C03632=1051.744,-43.846,429.339,170.450,30.999,155.847
C03633=1051.750,-43.595,429.326,170.452,31.001,155.847
C03634=1051.756,-43.346,429.313,170.454,31.002,155.847
C03635=1051.763,-43.096,429.301,170.456,31.005,155.847
C03636=1051.769,-42.847,429.288,170.458,31.006,155.848
C03637=1051.775,-42.597,429.275,170.460,31.008,155.848
C03638=1051.781,-42.347,429.262,170.461,31.009,155.848
C03639=1051.787,-42.098,429.249,170.463,31.011,155.848
C03640=1051.794,-41.848,429.237,170.465,31.012,155.848
C03641=1051.800,-41.599,429.224,170.467,31.014,155.848
C03642=1051.806,-41.349,429.211,170.469,31.015,155.849
C03643=1051.812,-41.100,429.198,170.471,31.017,155.849
C03644=1051.819,-40.849,429.185,170.473,31.018,155.849
C03645=1051.825,-40.600,429.172,170.475,31.020,155.849
C03646=1051.832,-40.351,429.160,170.476,31.021,155.849
C03647=1051.838,-40.101,429.147,170.478,31.023,155.849
C03648=1051.844,-39.852,429.133,170.480,31.024,155.850
C03649=1051.850,-39.602,429.121,170.482,31.026,155.850
C03650=1051.856,-39.353,429.108,170.484,31.028,155.850
C03651=1051.862,-39.103,429.095,170.486,31.030,155.850
C03652=1051.870,-38.853,429.082,170.488,31.031,155.850
C03653=1051.876,-38.604,429.069,170.490,31.033,155.850
C03654=1051.882,-38.354,429.056,170.491,31.034,155.851
C03655=1051.888,-38.105,429.043,170.493,31.036,155.851
C03656=1051.894,-37.855,429.030,170.495,31.037,155.851
C03657=1051.900,-37.606,429.017,170.497,31.039,155.851
C03658=1051.906,-37.357,429.004,170.499,31.041,155.851
C03659=1051.912,-37.107,428.991,170.501,31.042,155.852
C03660=1051.918,-36.856,428.977,170.503,31.044,155.852
C03661=1051.925,-36.607,428.964,170.504,31.046,155.852
C03662=1051.930,-36.357,428.951,170.506,31.048,155.852
C03663=1051.937,-36.108,428.938,170.508,31.049,155.852
C03664=1051.943,-35.859,428.925,170.509,31.051,155.853
C03665=1051.949,-35.609,428.912,170.511,31.053,155.853
C03666=1051.956,-35.359,428.899,170.513,31.054,155.853
C03667=1051.962,-35.080,428.884,170.516,31.056,155.853
C03668=1051.969,-34.799,428.869,170.518,31.058,155.853
C03669=1051.976,-34.519,428.855,170.519,31.060,155.854
C03670=1051.983,-34.239,428.840,170.521,31.062,155.854
C03671=1051.990,-33.989,428.826,170.523,31.063,155.854
C03672=1051.995,-33.739,428.813,170.525,31.065,155.854
C03673=1052.001,-33.490,428.800,170.527,31.067,155.854
C03674=1052.008,-33.241,428.786,170.529,31.068,155.855
C03675=1052.014,-32.991,428.773,170.531,31.070,155.855
C03676=1052.020,-32.741,428.760,170.533,31.072,155.855
C03677=1052.027,-32.492,428.747,170.534,31.074,155.855
C03678=1052.033,-32.242,428.734,170.536,31.075,155.855
C03679=1052.039,-31.993,428.720,170.538,31.077,155.856
C03680=1052.046,-31.743,428.707,170.540,31.079,155.856
C03681=1052.052,-31.494,428.694,170.542,31.080,155.856
C03682=1052.058,-31.244,428.681,170.544,31.082,155.856
C03683=1052.063,-30.994,428.667,170.546,31.084,155.856
C03684=1052.070,-30.744,428.653,170.547,31.085,155.857
C03685=1052.076,-30.495,428.640,170.548,31.087,155.857
C03686=1052.083,-30.246,428.627,170.550,31.088,155.857
C03687=1052.089,-29.997,428.614,170.552,31.091,155.857
C03688=1052.096,-29.747,428.600,170.554,31.092,155.857
C03689=1052.102,-29.497,428.587,170.556,31.094,155.858
C03690=1052.108,-29.247,428.574,170.558,31.096,155.858
C03691=1052.115,-28.997,428.561,170.560,31.097,155.858
C03692=1052.120,-28.748,428.547,170.561,31.099,155.858
C03693=1052.126,-28.499,428.533,170.563,31.101,155.858
C03694=1052.133,-28.249,428.520,170.565,31.102,155.859
C03695=1052.139,-27.999,428.507,170.567,31.104,155.859
C03696=1052.146,-27.750,428.493,170.569,31.106,155.859
C03697=1052.152,-27.501,428.480,170.571,31.108,155.859
C03698=1052.159,-27.251,428.466,170.573,31.109,155.859
C03699=1052.164,-27.001,428.453,170.575,31.111,155.860
C03700=1052.170,-26.752,428.439,170.575,31.113,155.860
C03701=1052.177,-26.502,428.426,170.577,31.114,155.860
C03702=1052.183,-26.253,428.412,170.579,31.116,155.860
C03703=1052.189,-26.003,428.398,170.581,31.118,155.861
C03704=1052.196,-25.753,428.385,170.583,31.120,155.861
C03705=1052.201,-25.504,428.371,170.585,31.121,155.861
C03706=1052.207,-25.254,428.358,170.587,31.124,155.861
C03707=1052.214,-25.004,428.344,170.589,31.125,155.861
C03708=1052.220,-24.755,428.330,170.590,31.127,155.862
C03709=1052.226,-24.506,428.317,170.592,31.129,155.862
C03710=1052.232,-24.256,428.304,170.594,31.130,155.862
C03711=1052.238,-24.006,428.289,170.595,31.132,155.862
C03712=1052.245,-23.757,428.275,170.597,31.134,155.863
C03713=1052.250,-23.508,428.262,170.599,31.136,155.863
C03714=1052.257,-23.258,428.248,170.601,31.137,155.863
C03715=1052.263,-23.009,428.235,170.603,31.140,155.863
C03716=1052.269,-22.758,428.220,170.604,31.141,155.863
C03717=1052.275,-22.509,428.207,170.606,31.143,155.864
C03718=1052.282,-22.260,428.194,170.608,31.145,155.864
C03719=1052.288,-22.010,428.179,170.610,31.147,155.864
C03720=1052.294,-21.761,428.166,170.612,31.148,155.864
C03721=1052.300,-21.511,428.152,170.613,31.150,155.865
C03722=1052.307,-21.261,428.138,170.615,31.152,155.865
C03723=1052.313,-21.012,428.125,170.616,31.154,155.865
C03724=1052.319,-20.762,428.111,170.618,31.155,155.865
C03725=1052.325,-20.513,428.097,170.620,31.158,155.866
C03726=1052.331,-20.264,428.083,170.622,31.159,155.866
C03727=1052.338,-20.014,428.069,170.624,31.161,155.866
C03728=1052.344,-19.764,428.056,170.626,31.163,155.866
C03729=1052.350,-19.515,428.041,170.628,31.165,155.866
C03730=1052.356,-19.265,428.028,170.630,31.166,155.867
C03731=1052.363,-18.984,428.012,170.631,31.169,155.867
C03732=1052.370,-18.703,427.996,170.633,31.171,155.867
C03733=1052.377,-18.422,427.981,170.635,31.173,155.867
C03734=1052.385,-18.141,427.965,170.637,31.175,155.868
C03735=1052.390,-17.892,427.951,170.639,31.176,155.868
C03736=1052.397,-17.643,427.938,170.641,31.179,155.868
C03737=1052.403,-17.393,427.923,170.643,31.180,155.868
C03738=1052.409,-17.144,427.910,170.644,31.182,155.869
C03739=1052.416,-16.894,427.895,170.645,31.184,155.869
C03740=1052.422,-16.645,427.882,170.647,31.186,155.869
C03741=1052.429,-16.395,427.868,170.649,31.187,155.869
C03742=1052.434,-16.146,427.854,170.651,31.189,155.870
C03743=1052.441,-15.896,427.840,170.653,31.191,155.870
C03744=1052.447,-15.646,427.826,170.655,31.193,155.870
C03745=1052.454,-15.397,427.812,170.657,31.195,155.870
C03746=1052.459,-15.147,427.798,170.658,31.197,155.870
C03747=1052.466,-14.897,427.784,170.660,31.198,155.871
C03748=1052.472,-14.648,427.770,170.661,31.200,155.871
C03749=1052.478,-14.398,427.755,170.663,31.202,155.871
C03750=1052.484,-14.149,427.741,170.665,31.204,155.871
C03751=1052.491,-13.899,427.727,170.667,31.206,155.872
C03752=1052.496,-13.650,427.713,170.669,31.208,155.872
C03753=1052.503,-13.400,427.699,170.671,31.210,155.872
C03754=1052.509,-13.151,427.685,170.672,31.212,155.872
C03755=1052.515,-12.901,427.670,170.673,31.214,155.873
C03756=1052.521,-12.652,427.657,170.675,31.215,155.873
C03757=1052.528,-12.402,427.642,170.677,31.217,155.873
C03758=1052.533,-12.153,427.628,170.679,31.219,155.873
C03759=1052.540,-11.903,427.614,170.681,31.221,155.874
C03760=1052.546,-11.654,427.600,170.683,31.223,155.874
C03761=1052.552,-11.404,427.585,170.685,31.225,155.874
C03762=1052.558,-11.155,427.572,170.685,31.227,155.874
C03763=1052.565,-10.905,427.557,170.687,31.229,155.875
C03764=1052.570,-10.655,427.543,170.689,31.231,155.875
C03765=1052.577,-10.406,427.529,170.691,31.232,155.875
C03766=1052.583,-10.157,427.514,170.693,31.234,155.875
C03767=1052.589,-9.907,427.500,170.695,31.237,155.876
C03768=1052.596,-9.658,427.486,170.697,31.238,155.876
C03769=1052.602,-9.408,427.471,170.698,31.240,155.876
C03770=1052.608,-9.158,427.457,170.699,31.242,155.876
C03771=1052.614,-8.909,427.443,170.701,31.244,155.877
C03772=1052.621,-8.659,427.428,170.703,31.246,155.877
C03773=1052.626,-8.410,427.414,170.705,31.248,155.877
C03774=1052.633,-8.160,427.400,170.707,31.250,155.877
C03775=1052.639,-7.912,427.386,170.708,31.251,155.878
C03776=1052.645,-7.662,427.371,170.710,31.253,155.878
C03777=1052.652,-7.412,427.356,170.712,31.256,155.878
C03778=1052.658,-7.163,427.342,170.713,31.257,155.878
C03779=1052.664,-6.913,427.328,170.715,31.259,155.879
C03780=1052.670,-6.663,427.313,170.717,31.261,155.879
C03781=1052.676,-6.414,427.299,170.718,31.263,155.879
C03782=1052.683,-6.164,427.285,170.720,31.265,155.879
C03783=1052.689,-5.915,427.270,170.722,31.267,155.880
C03784=1052.695,-5.665,427.255,170.724,31.268,155.880
C03785=1052.702,-5.416,427.240,170.726,31.271,155.880
C03786=1052.708,-5.167,427.227,170.727,31.273,155.880
C03787=1052.714,-4.917,427.212,170.729,31.275,155.881
C03788=1052.721,-4.667,427.197,170.730,31.276,155.881
C03789=1052.727,-4.418,427.184,170.732,31.278,155.881
C03790=1052.733,-4.168,427.169,170.734,31.280,155.881
C03791=1052.740,-3.919,427.154,170.736,31.282,155.882
C03792=1052.745,-3.670,427.140,170.738,31.284,155.882
C03793=1052.752,-3.420,427.126,170.739,31.286,155.882
C03794=1052.759,-3.170,427.111,170.740,31.288,155.883
C03795=1052.765,-2.888,427.094,170.742,31.290,155.883
C03796=1052.772,-2.606,427.078,170.744,31.292,155.883
C03797=1052.779,-2.323,427.062,170.746,31.294,155.883
C03798=1052.786,-2.040,427.045,170.749,31.297,155.884
C03799=1052.792,-1.791,427.030,170.750,31.299,155.884
C03800=1052.797,-1.541,427.014,170.752,31.301,155.884
C03801=1052.804,-1.292,426.999,170.753,31.303,155.885
C03802=1052.810,-1.043,426.985,170.755,31.305,155.885
C03803=1052.816,-0.793,426.970,170.757,31.307,155.885
C03804=1052.822,-0.543,426.956,170.758,31.309,155.885
C03805=1052.828,-0.294,426.941,170.760,31.311,155.886
C03806=1052.834,-0.044,426.926,170.762,31.313,155.886
C03807=1052.841,0.206,426.911,170.764,31.315,155.886
C03808=1052.846,0.455,426.897,170.765,31.318,155.887
C03809=1052.853,0.704,426.882,170.766,31.319,155.887
C03810=1052.859,0.954,426.867,170.768,31.321,155.887
C03811=1052.865,1.203,426.852,170.770,31.323,155.887
C03812=1052.871,1.452,426.837,170.772,31.325,155.888
C03813=1052.878,1.702,426.822,170.774,31.327,155.888
C03814=1052.883,1.951,426.808,170.775,31.329,155.888
C03815=1052.890,2.201,426.793,170.777,31.331,155.888
C03816=1052.896,2.450,426.778,170.778,31.334,155.889
C03817=1052.902,2.699,426.763,170.780,31.336,155.889
C03818=1052.908,2.949,426.748,170.782,31.337,155.889
C03819=1052.915,3.199,426.733,170.783,31.339,155.890
C03820=1052.920,3.449,426.718,170.785,31.341,155.890
C03821=1052.926,3.698,426.703,170.787,31.343,155.890
C03822=1052.933,3.947,426.688,170.789,31.345,155.890
C03823=1052.939,4.197,426.673,170.790,31.347,155.891
C03824=1052.945,4.447,426.658,170.792,31.350,155.891
C03825=1052.951,4.695,426.644,170.793,31.352,155.891
C03826=1052.958,4.945,426.629,170.795,31.354,155.892
C03827=1052.964,5.195,426.614,170.797,31.355,155.892
C03828=1052.970,5.444,426.599,170.798,31.357,155.892
C03829=1052.976,5.693,426.584,170.800,31.359,155.892
C03830=1052.982,5.943,426.569,170.802,31.361,155.893
C03831=1052.989,6.193,426.555,170.804,31.364,155.893
C03832=1052.995,6.443,426.539,170.805,31.366,155.893
C03833=1053.001,6.691,426.524,170.806,31.368,155.893
C03834=1053.007,6.941,426.509,170.808,31.370,155.894
C03835=1053.013,7.190,426.494,170.810,31.372,155.894
C03836=1053.020,7.440,426.479,170.812,31.374,155.894
C03837=1053.026,7.690,426.464,170.813,31.375,155.895
C03838=1053.033,7.939,426.449,170.815,31.377,155.895
C03839=1053.038,8.188,426.434,170.817,31.380,155.895
C03840=1053.045,8.437,426.419,170.819,31.382,155.895
C03841=1053.051,8.687,426.403,170.820,31.384,155.896
C03842=1053.057,8.937,426.388,170.821,31.386,155.896
C03843=1053.063,9.187,426.373,170.823,31.388,155.896
C03844=1053.070,9.436,426.358,170.825,31.390,155.897
C03845=1053.076,9.685,426.344,170.827,31.392,155.897
C03846=1053.082,9.934,426.328,170.829,31.394,155.897
C03847=1053.089,10.184,426.313,170.830,31.396,155.897
C03848=1053.095,10.434,426.298,170.832,31.398,155.898
C03849=1053.101,10.684,426.283,170.833,31.400,155.898
C03850=1053.107,10.933,426.267,170.835,31.402,155.898
C03851=1053.114,11.182,426.252,170.836,31.404,155.899
C03852=1053.120,11.431,426.237,170.838,31.406,155.899
C03853=1053.126,11.681,426.223,170.840,31.408,155.899
C03854=1053.133,11.930,426.207,170.842,31.410,155.899
C03855=1053.139,12.180,426.192,170.844,31.412,155.900
C03856=1053.145,12.429,426.176,170.845,31.414,155.900
C03857=1053.151,12.679,426.161,170.846,31.416,155.900
C03858=1053.158,12.928,426.146,170.848,31.418,155.900
C03859=1053.165,13.213,426.128,170.850,31.421,155.901
C03860=1053.172,13.497,426.111,170.852,31.423,155.901
C03861=1053.179,13.781,426.094,170.854,31.425,155.901
C03862=1053.186,14.066,426.077,170.856,31.427,155.902
C03863=1053.193,14.315,426.061,170.858,31.429,155.902
C03864=1053.199,14.565,426.046,170.859,31.431,155.902
C03865=1053.205,14.814,426.030,170.860,31.434,155.903
C03866=1053.211,15.064,426.015,170.862,31.436,155.903
C03867=1053.217,15.314,426.000,170.864,31.438,155.903
C03868=1053.224,15.563,425.984,170.865,31.440,155.904
C03869=1053.230,15.813,425.969,170.867,31.442,155.904
C03870=1053.236,16.062,425.953,170.869,31.444,155.904
C03871=1053.243,16.311,425.938,170.871,31.446,155.904
C03872=1053.248,16.561,425.923,170.872,31.448,155.905
C03873=1053.254,16.810,425.907,170.873,31.450,155.905
C03874=1053.260,17.060,425.892,170.875,31.452,155.905
C03875=1053.267,17.309,425.876,170.877,31.454,155.906
C03876=1053.273,17.558,425.861,170.878,31.456,155.906
C03877=1053.279,17.808,425.845,170.880,31.458,155.906
C03878=1053.285,18.057,425.830,170.882,31.461,155.906
C03879=1053.291,18.307,425.814,170.884,31.463,155.907
C03880=1053.298,18.556,425.799,170.885,31.465,155.907
C03881=1053.304,18.805,425.783,170.887,31.467,155.907
C03882=1053.310,19.055,425.767,170.888,31.469,155.908
C03883=1053.317,19.304,425.752,170.890,31.471,155.908
C03884=1053.322,19.554,425.736,170.891,31.473,155.908
C03885=1053.329,19.803,425.720,170.893,31.475,155.909
C03886=1053.335,20.053,425.706,170.895,31.477,155.909
C03887=1053.341,20.302,425.689,170.897,31.479,155.909
C03888=1053.347,20.552,425.673,170.898,31.481,155.909
C03889=1053.354,20.801,425.658,170.900,31.484,155.910
C03890=1053.360,21.051,425.642,170.901,31.486,155.910
C03891=1053.366,21.300,425.627,170.903,31.488,155.910
C03892=1053.372,21.550,425.611,170.904,31.490,155.911
C03893=1053.379,21.799,425.595,170.906,31.492,155.911
C03894=1053.384,22.049,425.579,170.908,31.494,155.911
C03895=1053.391,22.298,425.564,170.909,31.496,155.912
C03896=1053.397,22.548,425.548,170.911,31.498,155.912
C03897=1053.403,22.797,425.533,170.913,31.500,155.912
C03898=1053.409,23.046,425.516,170.914,31.502,155.913
C03899=1053.416,23.296,425.501,170.915,31.505,155.913
C03900=1053.422,23.545,425.485,170.917,31.507,155.913
C03901=1053.428,23.794,425.469,170.919,31.509,155.914
C03902=1053.434,24.044,425.454,170.921,31.511,155.914
C03903=1053.440,24.293,425.438,170.922,31.513,155.914
C03904=1053.447,24.542,425.422,170.924,31.515,155.914
C03905=1053.452,24.792,425.406,170.926,31.517,155.915
C03906=1053.459,25.041,425.391,170.928,31.519,155.915
C03907=1053.465,25.291,425.375,170.928,31.521,155.915
C03908=1053.471,25.540,425.358,170.930,31.524,155.916
C03909=1053.477,25.790,425.343,170.932,31.526,155.916
C03910=1053.483,26.039,425.327,170.933,31.528,155.916
C03911=1053.490,26.288,425.311,170.935,31.530,155.917
C03912=1053.496,26.538,425.295,170.937,31.532,155.917
C03913=1053.502,26.787,425.280,170.939,31.534,155.917
C03914=1053.508,27.037,425.264,170.940,31.536,155.917
C03915=1053.514,27.286,425.248,170.942,31.539,155.918
C03916=1053.521,27.535,425.232,170.943,31.541,155.918
C03917=1053.527,27.785,425.215,170.944,31.543,155.918
C03918=1053.533,28.035,425.200,170.946,31.545,155.919
C03919=1053.540,28.284,425.184,170.948,31.547,155.919
C03920=1053.546,28.533,425.168,170.950,31.549,155.919
C03921=1053.552,28.783,425.152,170.951,31.551,155.920
C03922=1053.558,29.032,425.136,170.953,31.554,155.920
C03923=1053.565,29.317,425.118,170.955,31.556,155.920
C03924=1053.573,29.603,425.099,170.956,31.558,155.921
C03925=1053.579,29.889,425.081,170.958,31.561,155.921
C03926=1053.586,30.175,425.063,170.960,31.564,155.921
C03927=1053.592,30.424,425.046,170.962,31.566,155.922
C03928=1053.598,30.673,425.030,170.963,31.568,155.922
C03929=1053.604,30.923,425.014,170.965,31.570,155.922
C03930=1053.611,31.172,424.998,170.967,31.573,155.923
C03931=1053.617,31.422,424.982,170.968,31.574,155.923
C03932=1053.623,31.672,424.966,170.969,31.577,155.923
C03933=1053.629,31.921,424.950,170.971,31.579,155.924
C03934=1053.635,32.170,424.933,170.973,31.581,155.924
C03935=1053.641,32.419,424.918,170.974,31.583,155.924
C03936=1053.647,32.669,424.902,170.976,31.585,155.925
C03937=1053.653,32.918,424.885,170.978,31.588,155.925
C03938=1053.660,33.168,424.869,170.979,31.589,155.925
C03939=1053.665,33.417,424.853,170.981,31.592,155.926
C03940=1053.672,33.665,424.836,170.983,31.594,155.926
C03941=1053.678,33.915,424.820,170.984,31.596,155.926
C03942=1053.684,34.164,424.804,170.985,31.598,155.927
C03943=1053.691,34.412,424.787,170.987,31.600,155.927
C03944=1053.697,34.662,424.771,170.989,31.602,155.927
C03945=1053.702,34.910,424.755,170.990,31.604,155.927
C03946=1053.709,35.159,424.740,170.992,31.607,155.928
C03947=1053.715,35.408,424.723,170.994,31.609,155.928
C03948=1053.722,35.658,424.706,170.995,31.611,155.928
C03949=1053.728,35.907,424.690,170.997,31.613,155.929
C03950=1053.734,36.157,424.674,170.998,31.615,155.929
C03951=1053.741,36.406,424.658,171.000,31.617,155.929
C03952=1053.747,36.655,424.642,171.001,31.620,155.930
C03953=1053.753,36.905,424.625,171.003,31.622,155.930
C03954=1053.759,37.155,424.609,171.005,31.624,155.930
C03955=1053.765,37.404,424.593,171.006,31.626,155.931
C03956=1053.771,37.653,424.576,171.008,31.628,155.931
C03957=1053.777,37.903,424.560,171.010,31.631,155.931
C03958=1053.784,38.152,424.543,171.011,31.633,155.932
C03959=1053.790,38.401,424.526,171.012,31.635,155.932
C03960=1053.796,38.651,424.510,171.014,31.637,155.932
C03961=1053.802,38.900,424.494,171.016,31.640,155.933
C03962=1053.808,39.149,424.478,171.017,31.642,155.933
C03963=1053.814,39.399,424.460,171.019,31.644,155.933
C03964=1053.820,39.648,424.444,171.021,31.646,155.934
C03965=1053.826,39.898,424.428,171.022,31.648,155.934
C03966=1053.832,40.147,424.412,171.024,31.650,155.934
C03967=1053.838,40.396,424.395,171.026,31.653,155.935
C03968=1053.845,40.646,424.378,171.026,31.655,155.935
C03969=1053.851,40.895,424.362,171.028,31.657,155.935
C03970=1053.857,41.144,424.345,171.030,31.659,155.936
C03971=1053.863,41.394,424.329,171.031,31.662,155.936
C03972=1053.870,41.643,424.312,171.033,31.664,155.936
C03973=1053.876,41.892,424.296,171.035,31.666,155.937
C03974=1053.882,42.142,424.279,171.036,31.668,155.937
C03975=1053.888,42.391,424.262,171.038,31.671,155.937
C03976=1053.894,42.641,424.246,171.040,31.673,155.938
C03977=1053.900,42.890,424.229,171.041,31.675,155.938
C03978=1053.906,43.140,424.213,171.042,31.677,155.938
C03979=1053.912,43.389,424.195,171.044,31.679,155.939
C03980=1053.918,43.638,424.179,171.046,31.681,155.939
C03981=1053.924,43.888,424.163,171.047,31.683,155.939
C03982=1053.931,44.136,424.146,171.049,31.686,155.940
C03983=1053.936,44.387,424.129,171.051,31.688,155.940
C03984=1053.943,44.636,424.112,171.052,31.691,155.940
C03985=1053.949,44.885,424.095,171.054,31.693,155.941
C03986=1053.955,45.134,424.079,171.056,31.695,155.941
C03987=1053.961,45.421,424.060,171.057,31.698,155.941
C03988=1053.969,45.707,424.040,171.058,31.700,155.942
C03989=1053.975,45.994,424.020,171.060,31.703,155.942
C03990=1053.982,46.281,424.001,171.062,31.705,155.943
C03991=1053.988,46.530,423.985,171.064,31.708,155.943
C03992=1053.994,46.780,423.967,171.066,31.710,155.943
C03993=1054.000,47.029,423.951,171.067,31.712,155.944
C03994=1054.006,47.278,423.934,171.069,31.715,155.944
C03995=1054.012,47.528,423.916,171.070,31.717,155.944
C03996=1054.019,47.777,423.899,171.071,31.719,155.945
C03997=1054.024,48.026,423.883,171.073,31.722,155.945
C03998=1054.031,48.275,423.866,171.075,31.724,155.945
C03999=1054.037,48.525,423.849,171.076,31.726,155.946
C04000=1054.043,48.774,423.832,171.078,31.728,155.946
C04001=1054.049,49.023,423.816,171.080,31.730,155.946
C04002=1054.055,49.273,423.798,171.081,31.733,155.947
C04003=1054.061,49.522,423.782,171.083,31.735,155.947
C04004=1054.067,49.771,423.765,171.085,31.737,155.947
C04005=1054.073,50.022,423.747,171.085,31.740,155.948
C04006=1054.079,50.270,423.730,171.087,31.742,155.948
C04007=1054.085,50.520,423.714,171.089,31.744,155.948
C04008=1054.091,50.769,423.696,171.090,31.746,155.949
C04009=1054.097,51.018,423.679,171.092,31.748,155.949
C04010=1054.104,51.268,423.663,171.094,31.751,155.950
C04011=1054.110,51.517,423.645,171.095,31.753,155.950
C04012=1054.115,51.767,423.629,171.097,31.755,155.950
C04013=1054.122,52.016,423.611,171.099,31.758,155.951
C04014=1054.128,52.265,423.594,171.099,31.760,155.951
C04015=1054.134,52.514,423.578,171.101,31.762,155.951
C04016=1054.141,52.764,423.560,171.103,31.764,155.952
C04017=1054.146,53.013,423.543,171.104,31.766,155.952
C04018=1054.153,53.263,423.526,171.106,31.768,155.952
C04019=1054.158,53.512,423.509,171.108,31.771,155.953
C04020=1054.165,53.761,423.492,171.109,31.773,155.953
C04021=1054.171,54.011,423.475,171.111,31.775,155.953
C04022=1054.177,54.260,423.457,171.113,31.778,155.954
C04023=1054.183,54.509,423.440,171.115,31.780,155.954
C04024=1054.189,54.759,423.424,171.115,31.782,155.954
C04025=1054.196,55.008,423.406,171.117,31.785,155.955
C04026=1054.202,55.257,423.389,171.119,31.787,155.955
C04027=1054.207,55.507,423.372,171.120,31.789,155.955
C04028=1054.214,55.756,423.355,171.122,31.791,155.956
C04029=1054.220,56.005,423.338,171.124,31.793,155.956
C04030=1054.226,56.255,423.320,171.125,31.796,155.956
C04031=1054.232,56.504,423.304,171.127,31.798,155.957
C04032=1054.239,56.753,423.286,171.129,31.800,155.957
C04033=1054.245,57.002,423.269,171.130,31.803,155.957
C04034=1054.251,57.252,423.251,171.131,31.805,155.958
C04035=1054.257,57.501,423.234,171.133,31.807,155.958
C04036=1054.263,57.751,423.217,171.134,31.809,155.958
C04037=1054.270,58.000,423.200,171.136,31.811,155.959
C04038=1054.276,58.249,423.182,171.138,31.813,155.959
C04039=1054.282,58.498,423.165,171.139,31.816,155.959
C04040=1054.288,58.748,423.148,171.141,31.818,155.960
C04041=1054.294,58.997,423.131,171.143,31.820,155.960
C04042=1054.301,59.247,423.114,171.144,31.822,155.960
C04043=1054.307,59.496,423.096,171.146,31.825,155.961
C04044=1054.313,59.745,423.079,171.147,31.827,155.961
C04045=1054.319,59.994,423.061,171.148,31.829,155.961
C04046=1054.325,60.244,423.045,171.150,31.831,155.962
C04047=1054.331,60.493,423.027,171.152,31.833,155.962
C04048=1054.338,60.743,423.010,171.153,31.835,155.962
C04049=1054.344,60.991,422.993,171.155,31.838,155.963
C04050=1054.350,61.241,422.975,171.157,31.840,155.963
C04051=1054.358,61.527,422.955,171.159,31.843,155.964
C04052=1054.365,61.811,422.935,171.161,31.845,155.964
C04053=1054.372,62.097,422.915,171.163,31.848,155.964
C04054=1054.379,62.383,422.896,171.163,31.850,155.965
C04055=1054.385,62.632,422.878,171.165,31.852,155.965
C04056=1054.392,62.881,422.861,171.167,31.855,155.965
C04057=1054.398,63.131,422.843,171.169,31.857,155.966
C04058=1054.404,63.380,422.826,171.170,31.859,155.966
C04059=1054.410,63.630,422.808,171.172,31.861,155.966
C04060=1054.416,63.878,422.791,171.174,31.864,155.967
C04061=1054.423,64.128,422.774,171.175,31.865,155.967
C04062=1054.429,64.377,422.756,171.177,31.868,155.967
C04063=1054.435,64.626,422.738,171.179,31.870,155.968
C04064=1054.442,64.876,422.721,171.180,31.872,155.968
C04065=1054.447,65.125,422.703,171.181,31.875,155.968
C04066=1054.453,65.375,422.685,171.183,31.877,155.969
C04067=1054.459,65.624,422.668,171.184,31.879,155.969
C04068=1054.466,65.873,422.651,171.186,31.881,155.970
C04069=1054.471,66.122,422.633,171.188,31.884,155.970
C04070=1054.478,66.371,422.614,171.189,31.886,155.970
C04071=1054.485,66.621,422.597,171.191,31.888,155.971
C04072=1054.490,66.870,422.579,171.193,31.891,155.971
C04073=1054.496,67.120,422.562,171.194,31.893,155.971
C04074=1054.502,67.368,422.545,171.196,31.895,155.972
C04075=1054.509,67.618,422.527,171.197,31.897,155.972
C04076=1054.515,67.868,422.509,171.198,31.899,155.972
C04077=1054.520,68.117,422.491,171.200,31.902,155.973
C04078=1054.527,68.366,422.474,171.202,31.904,155.973
C04079=1054.533,68.615,422.455,171.203,31.907,155.973
C04080=1054.539,68.864,422.438,171.205,31.909,155.974
C04081=1054.545,69.114,422.420,171.207,31.911,155.974
C04082=1054.551,69.363,422.403,171.208,31.913,155.974
C04083=1054.558,69.613,422.385,171.210,31.915,155.975
C04084=1054.564,69.862,422.367,171.212,31.918,155.975
C04085=1054.569,70.111,422.348,171.213,31.920,155.976
C04086=1054.576,70.360,422.331,171.214,31.923,155.976
C04087=1054.582,70.609,422.314,171.216,31.925,155.976
C04088=1054.588,70.859,422.296,171.217,31.927,155.977
C04089=1054.594,71.108,422.277,171.219,31.929,155.977
C04090=1054.600,71.357,422.259,171.221,31.932,155.977
C04091=1054.606,71.607,422.242,171.222,31.934,155.978
C04092=1054.612,71.857,422.224,171.224,31.937,155.978
C04093=1054.618,72.105,422.205,171.226,31.939,155.978
C04094=1054.624,72.355,422.187,171.227,31.941,155.979
C04095=1054.630,72.603,422.170,171.229,31.943,155.979
C04096=1054.637,72.853,422.152,171.231,31.946,155.980
C04097=1054.643,73.102,422.134,171.231,31.948,155.980
C04098=1054.648,73.351,422.116,171.233,31.950,155.980
C04099=1054.655,73.601,422.098,171.235,31.953,155.981
C04100=1054.661,73.850,422.080,171.236,31.955,155.981
C04101=1054.667,74.099,422.062,171.238,31.957,155.981
C04102=1054.673,74.348,422.043,171.240,31.959,155.982
C04103=1054.679,74.598,422.026,171.241,31.962,155.982
C04104=1054.685,74.848,422.008,171.243,31.964,155.982
C04105=1054.691,75.096,421.989,171.245,31.966,155.983
C04106=1054.697,75.346,421.971,171.246,31.968,155.983
C04107=1054.704,75.595,421.954,171.248,31.971,155.983
C04108=1054.710,75.844,421.936,171.249,31.973,155.984
C04109=1054.716,76.094,421.918,171.250,31.976,155.984
C04110=1054.722,76.343,421.899,171.252,31.978,155.985
C04111=1054.728,76.592,421.882,171.254,31.980,155.985
C04112=1054.734,76.842,421.864,171.255,31.982,155.985
C04113=1054.740,77.091,421.845,171.257,31.985,155.986
C04114=1054.747,77.340,421.827,171.259,31.987,155.986
C04115=1054.753,77.625,421.807,171.261,31.990,155.986
C04116=1054.760,77.911,421.786,171.262,31.992,155.987
C04117=1054.767,78.196,421.765,171.264,31.995,155.987
C04118=1054.774,78.481,421.744,171.266,31.997,155.988
C04119=1054.781,78.730,421.726,171.267,32.000,155.988
C04120=1054.786,78.979,421.708,171.269,32.002,155.988
C04121=1054.792,79.229,421.689,171.270,32.005,155.989
C04122=1054.798,79.478,421.670,171.272,32.007,155.989
C04123=1054.804,79.728,421.652,171.274,32.009,155.990
C04124=1054.810,79.976,421.634,171.275,32.011,155.990
C04125=1054.816,80.226,421.616,171.277,32.014,155.990
C04126=1054.823,80.475,421.597,171.279,32.016,155.991
C04127=1054.828,80.724,421.579,171.280,32.019,155.991
C04128=1054.834,80.973,421.560,171.282,32.021,155.991
C04129=1054.840,81.223,421.543,171.284,32.023,155.992
C04130=1054.847,81.472,421.524,171.284,32.026,155.992
C04131=1054.852,81.721,421.506,171.286,32.028,155.992
C04132=1054.859,81.970,421.488,171.288,32.031,155.993
C04133=1054.864,82.220,421.468,171.289,32.032,155.993
C04134=1054.871,82.469,421.450,171.291,32.035,155.994
C04135=1054.877,82.719,421.432,171.293,32.037,155.994
C04136=1054.883,82.967,421.414,171.294,32.040,155.994
C04137=1054.889,83.217,421.396,171.296,32.042,155.995
C04138=1054.894,83.466,421.376,171.298,32.044,155.995
C04139=1054.901,83.715,421.358,171.299,32.046,155.995
C04140=1054.906,83.965,421.340,171.301,32.049,155.996
C04141=1054.913,84.214,421.322,171.303,32.051,155.996
C04142=1054.919,84.463,421.303,171.303,32.054,155.997
C04143=1054.925,84.712,421.284,171.305,32.056,155.997
C04144=1054.931,84.962,421.266,171.307,32.058,155.997
C04145=1054.937,85.211,421.247,171.308,32.061,155.998
C04146=1054.943,85.459,421.229,171.310,32.063,155.998
C04147=1054.949,85.709,421.211,171.312,32.065,155.998
C04148=1054.955,85.959,421.192,171.313,32.067,155.999
C04149=1054.961,86.208,421.173,171.315,32.070,155.999
C04150=1054.968,86.457,421.154,171.317,32.072,155.999
C04151=1054.974,86.707,421.136,171.318,32.075,156.000
C04152=1054.979,86.955,421.117,171.320,32.077,156.000
C04153=1054.986,87.204,421.099,171.322,32.079,156.001
C04154=1054.992,87.454,421.080,171.323,32.081,156.001
C04155=1054.998,87.703,421.062,171.324,32.084,156.001
C04156=1055.004,87.953,421.043,171.326,32.086,156.002
C04157=1055.010,88.202,421.024,171.327,32.088,156.002
C04158=1055.017,88.451,421.006,171.329,32.091,156.002
C04159=1055.023,88.700,420.987,171.331,32.093,156.003
C04160=1055.029,88.949,420.969,171.333,32.095,156.003
C04161=1055.034,89.199,420.950,171.334,32.098,156.004
C04162=1055.041,89.448,420.932,171.336,32.100,156.004
C04163=1055.047,89.697,420.913,171.338,32.102,156.004
C04164=1055.054,89.946,420.894,171.339,32.104,156.005
C04165=1055.059,90.195,420.875,171.341,32.106,156.005
C04166=1055.066,90.445,420.856,171.343,32.109,156.005
C04167=1055.072,90.694,420.838,171.343,32.112,156.006
C04168=1055.078,90.943,420.819,171.345,32.114,156.006
C04169=1055.084,91.193,420.801,171.347,32.116,156.006
C04170=1055.089,91.442,420.782,171.348,32.118,156.007
C04171=1055.095,91.691,420.763,171.350,32.121,156.007
C04172=1055.101,91.940,420.744,171.352,32.123,156.008
C04173=1055.108,92.189,420.725,171.353,32.125,156.008
C04174=1055.113,92.439,420.706,171.355,32.128,156.008
C04175=1055.120,92.688,420.687,171.357,32.130,156.009
C04176=1055.125,92.937,420.668,171.358,32.133,156.009
C04177=1055.132,93.186,420.649,171.360,32.135,156.009
C04178=1055.137,93.436,420.630,171.362,32.137,156.010
C04179=1055.144,93.721,420.608,171.364,32.140,156.010
C04180=1055.152,94.006,420.587,171.365,32.143,156.011
C04181=1055.158,94.291,420.566,171.367,32.146,156.011
C04182=1055.165,94.576,420.544,171.369,32.148,156.012
C04183=1055.171,94.826,420.524,171.370,32.150,156.012
C04184=1055.177,95.075,420.506,171.372,32.153,156.012
C04185=1055.183,95.324,420.486,171.374,32.155,156.013
C04186=1055.189,95.573,420.468,171.375,32.158,156.013
C04187=1055.195,95.823,420.449,171.377,32.160,156.013
C04188=1055.202,96.072,420.430,171.379,32.162,156.014
C04189=1055.207,96.320,420.411,171.380,32.165,156.014
C04190=1055.213,96.570,420.392,171.382,32.167,156.014
C04191=1055.219,96.818,420.372,171.384,32.169,156.015
C04192=1055.225,97.068,420.354,171.385,32.171,156.015
C04193=1055.231,97.317,420.334,171.386,32.174,156.016
C04194=1055.238,97.566,420.316,171.388,32.177,156.016
C04195=1055.243,97.816,420.297,171.390,32.179,156.016
C04196=1055.249,98.065,420.277,171.391,32.181,156.017
C04197=1055.255,98.314,420.259,171.393,32.183,156.017
C04198=1055.261,98.563,420.239,171.395,32.186,156.018
C04199=1055.268,98.812,420.220,171.396,32.188,156.018
C04200=1055.274,99.061,420.201,171.398,32.190,156.018
C04201=1055.280,99.311,420.182,171.400,32.193,156.019
C04202=1055.286,99.560,420.163,171.401,32.195,156.019
C04203=1055.292,99.809,420.144,171.403,32.197,156.019
C04204=1055.299,100.059,420.124,171.405,32.200,156.020
C04205=1055.305,100.308,420.105,171.407,32.202,156.020
C04206=1055.311,100.557,420.086,171.408,32.204,156.020
C04207=1055.316,100.807,420.067,171.409,32.207,156.021
C04208=1055.323,101.055,420.047,171.411,32.209,156.021
C04209=1055.329,101.305,420.028,171.412,32.211,156.022
C04210=1055.335,101.554,420.009,171.414,32.214,156.022
C04211=1055.340,101.803,419.990,171.416,32.216,156.022
C04212=1055.347,102.052,419.970,171.417,32.219,156.023
C04213=1055.353,102.301,419.951,171.419,32.221,156.023
C04214=1055.358,102.551,419.932,171.421,32.223,156.024
C04215=1055.364,102.800,419.912,171.423,32.226,156.024
C04216=1055.370,103.049,419.893,171.424,32.228,156.024
C04217=1055.376,103.298,419.874,171.426,32.230,156.025
C04218=1055.382,103.547,419.854,171.428,32.233,156.025
C04219=1055.388,103.796,419.835,171.429,32.236,156.026
C04220=1055.394,104.045,419.815,171.431,32.238,156.026
C04221=1055.400,104.295,419.796,171.432,32.240,156.026
C04222=1055.406,104.544,419.777,171.433,32.242,156.027
C04223=1055.412,104.793,419.757,171.435,32.245,156.027
C04224=1055.418,105.042,419.738,171.437,32.247,156.027
C04225=1055.424,105.291,419.718,171.439,32.250,156.028
C04226=1055.430,105.540,419.699,171.440,32.252,156.028
C04227=1055.436,105.789,419.680,171.442,32.255,156.029
C04228=1055.443,106.039,419.660,171.444,32.257,156.029
C04229=1055.448,106.288,419.640,171.445,32.259,156.029
C04230=1055.454,106.537,419.620,171.447,32.262,156.030
C04231=1055.460,106.787,419.601,171.449,32.264,156.030
C04232=1055.466,107.035,419.581,171.451,32.267,156.030
C04233=1055.472,107.285,419.563,171.452,32.268,156.031
C04234=1055.478,107.533,419.543,171.454,32.271,156.031
C04235=1055.484,107.783,419.523,171.455,32.274,156.032
C04236=1055.490,108.032,419.503,171.456,32.276,156.032
C04237=1055.496,108.282,419.484,171.458,32.278,156.032
C04238=1055.502,108.531,419.464,171.460,32.280,156.033
C04239=1055.509,108.780,419.445,171.462,32.283,156.033
C04240=1055.515,109.028,419.425,171.463,32.285,156.034
C04241=1055.520,109.278,419.406,171.465,32.287,156.034
C04242=1055.526,109.527,419.386,171.467,32.290,156.034
C04243=1055.534,109.812,419.364,171.469,32.293,156.035
C04244=1055.541,110.097,419.342,171.471,32.295,156.035
C04245=1055.547,110.383,419.319,171.473,32.298,156.036
C04246=1055.555,110.668,419.296,171.475,32.301,156.036
C04247=1055.560,110.917,419.277,171.477,32.303,156.036
C04248=1055.566,111.166,419.257,171.478,32.306,156.037
C04249=1055.572,111.415,419.237,171.480,32.308,156.037
C04250=1055.579,111.665,419.217,171.481,32.310,156.038
C04251=1055.585,111.914,419.197,171.482,32.313,156.038
C04252=1055.590,112.163,419.178,171.484,32.315,156.038
C04253=1055.596,112.412,419.158,171.486,32.318,156.039
C04254=1055.602,112.661,419.138,171.488,32.320,156.039
C04255=1055.608,112.910,419.119,171.489,32.322,156.039
C04256=1055.615,113.160,419.099,171.491,32.325,156.040
C04257=1055.621,113.409,419.079,171.493,32.327,156.040
C04258=1055.627,113.657,419.059,171.495,32.329,156.041
C04259=1055.632,113.907,419.039,171.496,32.332,156.041
C04260=1055.638,114.156,419.020,171.498,32.334,156.041
C04261=1055.645,114.405,418.999,171.500,32.337,156.042
C04262=1055.650,114.655,418.980,171.502,32.339,156.042
C04263=1055.656,114.904,418.959,171.503,32.342,156.043
C04264=1055.662,115.153,418.939,171.505,32.344,156.043
C04265=1055.668,115.401,418.919,171.506,32.346,156.043
C04266=1055.674,115.650,418.900,171.507,32.349,156.044
C04267=1055.680,115.900,418.880,171.509,32.351,156.044
C04268=1055.685,116.149,418.859,171.511,32.354,156.045
C04269=1055.691,116.398,418.839,171.513,32.356,156.045
C04270=1055.697,116.647,418.819,171.514,32.359,156.045
C04271=1055.703,116.896,418.799,171.516,32.361,156.046
C04272=1055.709,117.145,418.779,171.518,32.364,156.046
C04273=1055.715,117.395,418.759,171.520,32.366,156.047
C04274=1055.721,117.644,418.739,171.521,32.368,156.047
C04275=1055.727,117.893,418.719,171.523,32.371,156.047
C04276=1055.732,118.142,418.699,171.525,32.374,156.048
C04277=1055.739,118.391,418.679,171.527,32.376,156.048
C04278=1055.745,118.640,418.659,171.528,32.378,156.049
C04279=1055.751,118.889,418.639,171.530,32.381,156.049
C04280=1055.756,119.138,418.618,171.532,32.383,156.049
C04281=1055.762,119.388,418.599,171.534,32.386,156.050
C04282=1055.768,119.637,418.578,171.534,32.388,156.050
C04283=1055.773,119.886,418.558,171.536,32.391,156.051
C04284=1055.779,120.135,418.538,171.538,32.393,156.051
C04285=1055.785,120.384,418.518,171.540,32.395,156.051
C04286=1055.792,120.633,418.498,171.541,32.398,156.052
C04287=1055.797,120.882,418.477,171.543,32.400,156.052
C04288=1055.803,121.131,418.457,171.545,32.403,156.053
C04289=1055.810,121.381,418.437,171.547,32.405,156.053
C04290=1055.816,121.630,418.417,171.548,32.407,156.053
C04291=1055.821,121.879,418.396,171.550,32.410,156.054
C04292=1055.827,122.128,418.376,171.552,32.413,156.054
C04293=1055.834,122.377,418.356,171.554,32.415,156.055
C04294=1055.839,122.626,418.335,171.555,32.417,156.055
C04295=1055.845,122.875,418.316,171.557,32.420,156.055
C04296=1055.852,123.125,418.295,171.559,32.422,156.056
C04297=1055.857,123.374,418.275,171.561,32.424,156.056
C04298=1055.863,123.622,418.255,171.562,32.427,156.057
C04299=1055.869,123.872,418.234,171.563,32.430,156.057
C04300=1055.876,124.120,418.214,171.565,32.432,156.057
C04301=1055.881,124.369,418.193,171.567,32.434,156.058
C04302=1055.888,124.619,418.173,171.569,32.437,156.058
C04303=1055.894,124.868,418.153,171.570,32.439,156.059
C04304=1055.899,125.117,418.132,171.572,32.441,156.059
C04305=1055.905,125.366,418.112,171.574,32.444,156.059
C04306=1055.911,125.615,418.092,171.576,32.447,156.060
C04307=1055.918,125.900,418.068,171.578,32.449,156.060
C04308=1055.925,126.185,418.045,171.580,32.452,156.061
C04309=1055.932,126.471,418.021,171.582,32.454,156.061
C04310=1055.939,126.756,417.998,171.584,32.457,156.061
C04311=1055.945,127.005,417.978,171.586,32.460,156.062
C04312=1055.951,127.254,417.958,171.587,32.462,156.062
C04313=1055.957,127.503,417.937,171.589,32.465,156.063
C04314=1055.963,127.752,417.916,171.591,32.467,156.063
C04315=1055.970,128.001,417.896,171.593,32.469,156.064
C04316=1055.975,128.250,417.875,171.595,32.472,156.064
C04317=1055.981,128.500,417.855,171.596,32.474,156.064
C04318=1055.988,128.748,417.834,171.597,32.476,156.065
C04319=1055.993,128.997,417.814,171.599,32.479,156.065
C04320=1056.000,129.247,417.793,171.601,32.481,156.065
C04321=1056.006,129.495,417.774,171.603,32.484,156.066
C04322=1056.012,129.745,417.752,171.605,32.486,156.066
C04323=1056.018,129.993,417.732,171.606,32.488,156.067
C04324=1056.024,130.243,417.712,171.608,32.491,156.067
C04325=1056.030,130.492,417.691,171.610,32.493,156.067
C04326=1056.036,130.741,417.670,171.612,32.495,156.068
C04327=1056.042,130.990,417.649,171.614,32.498,156.068
C04328=1056.048,131.240,417.629,171.615,32.501,156.069
C04329=1056.055,131.488,417.608,171.617,32.503,156.069
C04330=1056.060,131.738,417.588,171.619,32.505,156.069
C04331=1056.066,131.986,417.568,171.621,32.508,156.070
C04332=1056.072,132.235,417.546,171.623,32.510,156.070
C04333=1056.078,132.485,417.525,171.624,32.512,156.071
C04334=1056.084,132.733,417.505,171.626,32.515,156.071
C04335=1056.090,132.983,417.484,171.628,32.518,156.071
C04336=1056.095,133.232,417.463,171.630,32.520,156.072
C04337=1056.102,133.481,417.442,171.631,32.523,156.072
C04338=1056.107,133.730,417.422,171.633,32.525,156.073
C04339=1056.114,133.979,417.400,171.634,32.527,156.073
C04340=1056.120,134.228,417.380,171.636,32.530,156.073
C04341=1056.125,134.476,417.359,171.638,32.532,156.074
C04342=1056.132,134.726,417.338,171.640,32.535,156.074
C04343=1056.137,134.974,417.317,171.642,32.538,156.075
C04344=1056.143,135.224,417.296,171.643,32.540,156.075
C04345=1056.149,135.472,417.276,171.645,32.542,156.075
C04346=1056.155,135.722,417.255,171.647,32.545,156.076
C04347=1056.161,135.971,417.233,171.649,32.547,156.076
C04348=1056.167,136.220,417.213,171.651,32.549,156.077
C04349=1056.173,136.469,417.192,171.653,32.552,156.077
C04350=1056.179,136.719,417.171,171.654,32.554,156.077
C04351=1056.185,136.967,417.150,171.656,32.557,156.078
C04352=1056.191,137.217,417.129,171.658,32.560,156.078
C04353=1056.197,137.466,417.108,171.660,32.562,156.079
C04354=1056.203,137.715,417.088,171.662,32.564,156.079
C04355=1056.209,137.964,417.066,171.664,32.567,156.080
C04356=1056.215,138.212,417.045,171.665,32.569,156.080
C04357=1056.221,138.462,417.024,171.667,32.572,156.080
C04358=1056.227,138.710,417.003,171.668,32.574,156.081
C04359=1056.233,138.960,416.982,171.670,32.577,156.081
C04360=1056.239,139.209,416.961,171.672,32.579,156.082
C04361=1056.245,139.458,416.939,171.674,32.582,156.082
C04362=1056.251,139.707,416.919,171.676,32.584,156.082
C04363=1056.257,139.956,416.898,171.677,32.587,156.083
C04364=1056.263,140.205,416.876,171.679,32.589,156.083
C04365=1056.268,140.454,416.856,171.681,32.592,156.084
C04366=1056.274,140.703,416.834,171.683,32.594,156.084
C04367=1056.280,140.952,416.813,171.685,32.597,156.084
C04368=1056.286,141.201,416.791,171.687,32.599,156.085
C04369=1056.291,141.450,416.771,171.688,32.602,156.085
C04370=1056.298,141.699,416.749,171.690,32.604,156.086
C04371=1056.305,141.984,416.724,171.692,32.607,156.086
C04372=1056.311,142.269,416.701,171.695,32.610,156.087
C04373=1056.318,142.554,416.676,171.697,32.613,156.087
C04374=1056.325,142.839,416.652,171.699,32.616,156.088
C04375=1056.331,143.088,416.630,171.701,32.618,156.088
C04376=1056.337,143.337,416.610,171.703,32.621,156.088
C04377=1056.343,143.586,416.588,171.704,32.623,156.089
C04378=1056.348,143.835,416.567,171.706,32.626,156.089
C04379=1056.354,144.084,416.545,171.708,32.628,156.090
C04380=1056.361,144.333,416.524,171.710,32.631,156.090
C04381=1056.366,144.582,416.503,171.711,32.633,156.090
C04382=1056.373,144.831,416.482,171.713,32.636,156.091
C04383=1056.379,145.080,416.460,171.715,32.638,156.091
C04384=1056.385,145.329,416.439,171.717,32.641,156.092
C04385=1056.391,145.578,416.417,171.718,32.643,156.092
C04386=1056.396,145.827,416.396,171.720,32.646,156.093
C04387=1056.402,146.076,416.374,171.722,32.648,156.093
C04388=1056.409,146.325,416.353,171.724,32.650,156.093
C04389=1056.414,146.574,416.332,171.726,32.653,156.094
C04390=1056.420,146.823,416.311,171.728,32.656,156.094
C04391=1056.426,147.073,416.289,171.730,32.658,156.095
C04392=1056.432,147.322,416.267,171.732,32.661,156.095
C04393=1056.438,147.570,416.246,171.734,32.663,156.096
C04394=1056.444,147.820,416.224,171.735,32.666,156.096
C04395=1056.450,148.069,416.203,171.737,32.668,156.096
C04396=1056.456,148.317,416.182,171.739,32.670,156.097
C04397=1056.462,148.566,416.160,171.741,32.673,156.097
C04398=1056.468,148.816,416.138,171.743,32.676,156.098
C04399=1056.474,149.064,416.117,171.745,32.678,156.098
C04400=1056.480,149.313,416.095,171.747,32.681,156.098
C04401=1056.485,149.563,416.073,171.749,32.683,156.099
C04402=1056.491,149.811,416.052,171.751,32.686,156.099
C04403=1056.497,150.061,416.030,171.752,32.689,156.100
C04404=1056.503,150.309,416.008,171.754,32.691,156.100
C04405=1056.509,150.558,415.987,171.756,32.694,156.101
C04406=1056.515,150.807,415.965,171.758,32.696,156.101
C04407=1056.521,151.056,415.943,171.760,32.699,156.101
C04408=1056.527,151.306,415.921,171.761,32.701,156.102
C04409=1056.532,151.554,415.900,171.763,32.704,156.102
C04410=1056.538,151.803,415.878,171.765,32.707,156.103
C04411=1056.545,152.053,415.857,171.767,32.709,156.103
C04412=1056.551,152.300,415.835,171.769,32.711,156.103
C04413=1056.557,152.550,415.813,171.771,32.714,156.104
C04414=1056.562,152.799,415.791,171.772,32.716,156.104
C04415=1056.568,153.048,415.769,171.774,32.719,156.105
C04416=1056.574,153.297,415.748,171.776,32.721,156.105
C04417=1056.580,153.546,415.726,171.778,32.724,156.106
C04418=1056.586,153.795,415.704,171.780,32.727,156.106
C04419=1056.592,154.044,415.682,171.782,32.729,156.107
C04420=1056.597,154.293,415.660,171.784,32.732,156.107
C04421=1056.604,154.542,415.639,171.786,32.734,156.107
C04422=1056.610,154.790,415.616,171.788,32.737,156.108
C04423=1056.616,155.040,415.595,171.790,32.740,156.108
C04424=1056.622,155.289,415.573,171.792,32.742,156.109
C04425=1056.627,155.538,415.551,171.794,32.745,156.109
C04426=1056.634,155.786,415.529,171.796,32.747,156.110
C04427=1056.639,156.036,415.507,171.798,32.750,156.110
C04428=1056.645,156.285,415.485,171.800,32.753,156.110
C04429=1056.651,156.533,415.463,171.801,32.755,156.111
C04430=1056.657,156.782,415.441,171.803,32.758,156.111
C04431=1056.663,157.032,415.419,171.805,32.760,156.112
C04432=1056.669,157.280,415.397,171.807,32.763,156.112
C04433=1056.675,157.530,415.375,171.809,32.765,156.113
C04434=1056.681,157.779,415.353,171.811,32.768,156.113
C04435=1056.687,158.063,415.328,171.813,32.771,156.114
C04436=1056.694,158.348,415.303,171.816,32.774,156.114
C04437=1056.701,158.632,415.277,171.818,32.777,156.115
C04438=1056.707,158.917,415.252,171.819,32.780,156.115
C04439=1056.714,159.166,415.230,171.821,32.782,156.115
C04440=1056.720,159.415,415.208,171.823,32.785,156.116
C04441=1056.725,159.664,415.185,171.825,32.787,156.116
C04442=1056.732,159.913,415.163,171.827,32.790,156.117
C04443=1056.737,160.161,415.141,171.829,32.792,156.117
C04444=1056.743,160.411,415.119,171.831,32.795,156.118
C04445=1056.749,160.660,415.098,171.833,32.798,156.118
C04446=1056.755,160.909,415.075,171.835,32.800,156.118
C04447=1056.761,161.157,415.052,171.837,32.803,156.119
C04448=1056.767,161.407,415.030,171.839,32.806,156.119
C04449=1056.772,161.655,415.008,171.841,32.809,156.120
C04450=1056.778,161.904,414.986,171.843,32.811,156.120
C04451=1056.784,162.153,414.963,171.845,32.814,156.121
C04452=1056.789,162.403,414.941,171.847,32.816,156.121
C04453=1056.796,162.651,414.918,171.849,32.819,156.122
C04454=1056.801,162.899,414.896,171.851,32.822,156.122
C04455=1056.806,163.149,414.874,171.853,32.825,156.123
C04456=1056.812,163.398,414.851,171.855,32.827,156.123
C04457=1056.818,163.647,414.829,171.856,32.830,156.123
C04458=1056.824,163.896,414.806,171.858,32.833,156.124
C04459=1056.830,164.145,414.783,171.860,32.835,156.124
C04460=1056.835,164.394,414.761,171.862,32.838,156.125
C04461=1056.841,164.642,414.739,171.864,32.841,156.125
C04462=1056.847,164.891,414.716,171.866,32.843,156.126
C04463=1056.852,165.140,414.693,171.868,32.846,156.126
C04464=1056.858,165.389,414.671,171.870,32.849,156.127
C04465=1056.864,165.638,414.648,171.872,32.851,156.127
C04466=1056.870,165.887,414.625,171.874,32.854,156.128
C04467=1056.875,166.136,414.603,171.876,32.857,156.128
C04468=1056.881,166.385,414.580,171.878,32.860,156.129
C04469=1056.887,166.633,414.558,171.880,32.862,156.129
C04470=1056.893,166.882,414.535,171.882,32.865,156.129
C04471=1056.898,167.132,414.513,171.884,32.867,156.130
C04472=1056.904,167.381,414.490,171.886,32.870,156.130
C04473=1056.910,167.629,414.468,171.888,32.873,156.131
C04474=1056.916,167.878,414.445,171.890,32.876,156.131
C04475=1056.922,168.127,414.422,171.892,32.878,156.132
C04476=1056.927,168.376,414.400,171.894,32.881,156.132
C04477=1056.934,168.625,414.377,171.896,32.883,156.133
C04478=1056.939,168.874,414.354,171.898,32.887,156.133
C04479=1056.945,169.123,414.331,171.900,32.889,156.134
C04480=1056.951,169.372,414.308,171.902,32.892,156.134
C04481=1056.957,169.621,414.286,171.903,32.894,156.134
C04482=1056.963,169.869,414.263,171.906,32.897,156.135
C04483=1056.968,170.119,414.241,171.908,32.900,156.135
C04484=1056.974,170.368,414.218,171.910,32.903,156.136
C04485=1056.980,170.617,414.195,171.912,32.905,156.136
C04486=1056.986,170.865,414.172,171.914,32.908,156.137
C04487=1056.992,171.114,414.150,171.916,32.910,156.137
C04488=1056.998,171.363,414.127,171.918,32.914,156.138
C04489=1057.004,171.612,414.104,171.920,32.916,156.138
C04490=1057.009,171.861,414.081,171.922,32.919,156.139
C04491=1057.015,172.110,414.058,171.924,32.921,156.139
C04492=1057.022,172.358,414.036,171.926,32.924,156.139
C04493=1057.027,172.607,414.013,171.928,32.926,156.140
C04494=1057.033,172.856,413.990,171.930,32.930,156.140
C04495=1057.039,173.105,413.967,171.932,32.932,156.141
C04496=1057.044,173.354,413.944,171.934,32.935,156.141
C04497=1057.050,173.603,413.921,171.936,32.937,156.142
C04498=1057.057,173.851,413.899,171.938,32.940,156.142
C04499=1057.063,174.136,413.872,171.941,32.943,156.143
C04500=1057.070,174.420,413.846,171.943,32.946,156.143
C04501=1057.077,174.704,413.820,171.945,32.949,156.144
C04502=1057.083,174.988,413.793,171.948,32.953,156.144
C04503=1057.090,175.237,413.771,171.950,32.955,156.145
C04504=1057.096,175.486,413.748,171.952,32.958,156.145
C04505=1057.102,175.736,413.725,171.954,32.960,156.146
C04506=1057.108,175.984,413.702,171.956,32.963,156.146
C04507=1057.113,176.233,413.679,171.958,32.966,156.147
C04508=1057.119,176.482,413.656,171.960,32.969,156.147
C04509=1057.125,176.731,413.633,171.962,32.971,156.148
C04510=1057.132,176.979,413.610,171.964,32.974,156.148
C04511=1057.137,177.228,413.587,171.967,32.977,156.148
C04512=1057.144,177.478,413.563,171.969,32.980,156.149
C04513=1057.149,177.726,413.541,171.971,32.982,156.149
C04514=1057.155,177.975,413.518,171.973,32.985,156.150
C04515=1057.161,178.224,413.494,171.975,32.987,156.150
C04516=1057.167,178.473,413.471,171.977,32.991,156.151
C04517=1057.173,178.721,413.448,171.979,32.993,156.151
C04518=1057.180,178.971,413.425,171.981,32.996,156.152
C04519=1057.185,179.220,413.402,171.983,32.998,156.152
C04520=1057.191,179.468,413.379,171.986,33.001,156.153
C04521=1057.197,179.717,413.356,171.988,33.004,156.153
C04522=1057.203,179.966,413.333,171.990,33.007,156.154
C04523=1057.210,180.215,413.309,171.992,33.009,156.154
C04524=1057.215,180.464,413.286,171.994,33.012,156.154
C04525=1057.221,180.712,413.263,171.996,33.014,156.155
C04526=1057.227,180.961,413.240,171.998,33.017,156.155
C04527=1057.233,181.210,413.216,172.000,33.020,156.156
C04528=1057.240,181.459,413.194,172.003,33.023,156.156
C04529=1057.246,181.708,413.171,172.005,33.025,156.157
C04530=1057.252,181.956,413.147,172.007,33.028,156.157
C04531=1057.258,182.206,413.124,172.009,33.031,156.158
C04532=1057.264,182.454,413.100,172.011,33.033,156.158
C04533=1057.270,182.703,413.077,172.013,33.036,156.159
C04534=1057.276,182.952,413.054,172.015,33.039,156.159
C04535=1057.282,183.201,413.030,172.018,33.042,156.160
C04536=1057.288,183.450,413.007,172.020,33.044,156.160
C04537=1057.294,183.699,412.983,172.022,33.047,156.160
C04538=1057.300,183.947,412.960,172.024,33.049,156.161
C04539=1057.306,184.196,412.937,172.026,33.053,156.161
C04540=1057.313,184.445,412.913,172.028,33.055,156.162
C04541=1057.318,184.694,412.890,172.031,33.058,156.162
C04542=1057.324,184.943,412.866,172.033,33.061,156.163
C04543=1057.330,185.191,412.842,172.035,33.064,156.163
C04544=1057.335,185.440,412.819,172.037,33.067,156.164
C04545=1057.341,185.689,412.795,172.039,33.069,156.164
C04546=1057.347,185.938,412.772,172.041,33.072,156.165
C04547=1057.352,186.187,412.748,172.043,33.075,156.165
C04548=1057.358,186.436,412.725,172.046,33.078,156.166
C04549=1057.364,186.684,412.701,172.048,33.081,156.166
C04550=1057.370,186.933,412.676,172.050,33.084,156.167
C04551=1057.376,187.182,412.653,172.052,33.087,156.167
C04552=1057.381,187.431,412.629,172.054,33.090,156.168
C04553=1057.387,187.679,412.605,172.056,33.093,156.168
C04554=1057.393,187.929,412.582,172.059,33.095,156.169
C04555=1057.399,188.177,412.558,172.061,33.098,156.169
C04556=1057.405,188.425,412.534,172.063,33.101,156.170
C04557=1057.410,188.675,412.510,172.065,33.104,156.170
C04558=1057.416,188.924,412.487,172.067,33.107,156.171
C04559=1057.422,189.172,412.462,172.069,33.110,156.171
C04560=1057.428,189.421,412.439,172.072,33.112,156.172
C04561=1057.433,189.670,412.415,172.074,33.116,156.172
C04562=1057.439,189.919,412.391,172.076,33.118,156.173
C04563=1057.446,190.202,412.363,172.078,33.122,156.173
C04564=1057.452,190.486,412.336,172.081,33.125,156.174
C04565=1057.459,190.770,412.309,172.083,33.128,156.175
C04566=1057.466,191.054,412.282,172.086,33.131,156.175
C04567=1057.472,191.302,412.258,172.088,33.135,156.176
C04568=1057.478,191.552,412.234,172.090,33.137,156.176
C04569=1057.483,191.800,412.211,172.093,33.140,156.177
C04570=1057.489,192.049,412.186,172.095,33.143,156.177
C04571=1057.495,192.298,412.162,172.097,33.146,156.178
C04572=1057.501,192.547,412.138,172.099,33.149,156.178
C04573=1057.507,192.796,412.114,172.101,33.152,156.179
C04574=1057.513,193.044,412.090,172.104,33.155,156.179
C04575=1057.519,193.292,412.066,172.106,33.158,156.180
C04576=1057.524,193.542,412.041,172.108,33.161,156.180
C04577=1057.530,193.790,412.018,172.110,33.163,156.181
C04578=1057.536,194.040,411.994,172.113,33.166,156.181
C04579=1057.542,194.288,411.970,172.115,33.170,156.182
C04580=1057.548,194.538,411.946,172.117,33.172,156.182
C04581=1057.554,194.786,411.922,172.119,33.175,156.183
C04582=1057.559,195.034,411.898,172.121,33.178,156.183
C04583=1057.566,195.283,411.874,172.124,33.181,156.184
C04584=1057.571,195.532,411.849,172.126,33.184,156.184
C04585=1057.578,195.781,411.825,172.128,33.187,156.185
C04586=1057.583,196.030,411.801,172.130,33.190,156.185
C04587=1057.590,196.278,411.777,172.133,33.192,156.186
C04588=1057.595,196.527,411.753,172.135,33.196,156.186
C04589=1057.602,196.776,411.729,172.137,33.198,156.187
C04590=1057.607,197.025,411.705,172.139,33.201,156.187
C04591=1057.614,197.273,411.680,172.142,33.204,156.188
C04592=1057.619,197.522,411.656,172.144,33.207,156.188
C04593=1057.626,197.771,411.632,172.146,33.210,156.189
C04594=1057.631,198.019,411.607,172.149,33.213,156.189
C04595=1057.638,198.268,411.583,172.151,33.216,156.190
C04596=1057.643,198.517,411.559,172.153,33.219,156.190
C04597=1057.649,198.766,411.534,172.155,33.222,156.191
C04598=1057.655,199.014,411.511,172.158,33.225,156.191
C04599=1057.661,199.263,411.485,172.160,33.227,156.192
C04600=1057.668,199.512,411.461,172.162,33.230,156.192
C04601=1057.673,199.761,411.437,172.165,33.234,156.193
C04602=1057.680,200.009,411.413,172.167,33.236,156.193
C04603=1057.685,200.258,411.389,172.169,33.239,156.194
C04604=1057.692,200.507,411.365,172.171,33.242,156.194
C04605=1057.697,200.755,411.340,172.174,33.245,156.195
C04606=1057.703,201.004,411.315,172.176,33.248,156.195
C04607=1057.710,201.253,411.291,172.178,33.251,156.196
C04608=1057.715,201.502,411.267,172.181,33.254,156.196
C04609=1057.722,201.750,411.242,172.183,33.257,156.197
C04610=1057.728,202.000,411.218,172.185,33.260,156.197
C04611=1057.733,202.248,411.193,172.188,33.263,156.198
C04612=1057.740,202.497,411.168,172.190,33.266,156.199
C04613=1057.745,202.745,411.144,172.192,33.269,156.199
C04614=1057.752,202.994,411.120,172.194,33.272,156.200
C04615=1057.757,203.242,411.095,172.197,33.275,156.200
C04616=1057.763,203.492,411.070,172.199,33.278,156.201
C04617=1057.769,203.740,411.045,172.201,33.281,156.201
C04618=1057.775,203.989,411.020,172.204,33.284,156.202
C04619=1057.781,204.238,410.996,172.206,33.287,156.202
C04620=1057.786,204.486,410.971,172.208,33.290,156.203
C04621=1057.792,204.735,410.946,172.211,33.293,156.203
C04622=1057.798,204.983,410.922,172.214,33.296,156.204
C04623=1057.804,205.232,410.897,172.216,33.299,156.204
C04624=1057.810,205.481,410.872,172.219,33.303,156.205
C04625=1057.816,205.730,410.848,172.221,33.306,156.206
C04626=1057.822,205.978,410.822,172.223,33.309,156.206
C04627=1057.847,207.029,410.718,172.415,33.397,156.218
C04628=1057.853,207.263,410.694,172.417,33.400,156.218
C04629=1057.859,207.498,410.669,172.419,33.404,156.219
C04630=1057.864,207.733,410.645,172.421,33.408,156.220
C04631=1057.870,207.967,410.621,172.422,33.411,156.220
C04632=1057.876,208.202,410.597,172.424,33.415,156.221
C04633=1057.882,208.436,410.573,172.426,33.419,156.222
C04634=1057.889,208.671,410.548,172.428,33.422,156.222
C04635=1057.894,208.906,410.524,172.429,33.426,156.223
C04636=1057.900,209.154,410.498,172.431,33.430,156.224
C04637=1057.906,209.402,410.472,172.433,33.434,156.225
C04638=1057.913,209.651,410.447,172.435,33.438,156.225
C04639=1057.918,209.899,410.420,172.437,33.442,156.226
C04640=1057.925,210.149,410.394,172.439,33.446,156.227
C04641=1057.931,210.397,410.369,172.442,33.450,156.228
C04642=1057.937,210.646,410.342,172.444,33.453,156.228
C04643=1057.943,210.894,410.317,172.446,33.457,156.229
C04644=1057.950,211.142,410.291,172.447,33.461,156.230
C04645=1057.955,211.391,410.265,172.449,33.465,156.230
C04646=1057.962,211.639,410.239,172.451,33.469,156.231
C04647=1057.969,211.889,410.213,172.453,33.473,156.232
C04648=1057.974,212.137,410.187,172.455,33.477,156.233
C04649=1057.981,212.386,410.161,172.457,33.481,156.233
C04650=1057.987,212.634,410.135,172.459,33.484,156.234
C04651=1057.993,212.883,410.109,172.461,33.489,156.235
C04652=1057.999,213.131,410.083,172.463,33.492,156.236
C04653=1058.005,213.381,410.057,172.465,33.496,156.236
C04654=1058.012,213.629,410.031,172.467,33.500,156.237
C04655=1058.017,213.877,410.004,172.469,33.504,156.238
C04656=1058.024,214.126,409.979,172.471,33.508,156.239
C04657=1058.029,214.374,409.952,172.473,33.512,156.239
C04658=1058.036,214.622,409.926,172.475,33.515,156.240
C04659=1058.042,214.872,409.900,172.477,33.520,156.241
C04660=1058.049,215.120,409.874,172.479,33.523,156.242
C04661=1058.054,215.368,409.847,172.481,33.528,156.242
C04662=1058.061,215.617,409.822,172.483,33.531,156.243
C04663=1058.066,215.865,409.795,172.485,33.535,156.244
C04664=1058.073,216.114,409.769,172.487,33.539,156.245
C04665=1058.079,216.363,409.743,172.489,33.543,156.245
C04666=1058.085,216.611,409.717,172.491,33.547,156.246
C04667=1058.091,216.859,409.690,172.493,33.551,156.247
C04668=1058.098,217.109,409.665,172.496,33.554,156.247
C04669=1058.104,217.357,409.638,172.498,33.558,156.248
C04670=1058.110,217.605,409.611,172.500,33.562,156.249
C04671=1058.116,217.853,409.585,172.502,33.566,156.250
C04672=1058.122,218.103,409.558,172.504,33.570,156.250
C04673=1058.129,218.351,409.533,172.505,33.574,156.251
C04674=1058.134,218.600,409.506,172.507,33.577,156.252
C04675=1058.142,218.848,409.480,172.509,33.581,156.253
C04676=1058.147,219.097,409.453,172.511,33.585,156.253
C04677=1058.154,219.345,409.427,172.513,33.589,156.254
C04678=1058.160,219.594,409.401,172.515,33.593,156.255
C04679=1058.166,219.842,409.375,172.517,33.596,156.255
C04680=1058.172,220.091,409.348,172.520,33.601,156.256
C04681=1058.179,220.340,409.321,172.522,33.604,156.257
C04682=1058.185,220.588,409.295,172.524,33.608,156.258
C04683=1058.191,220.836,409.268,172.526,33.612,156.258
C04684=1058.197,221.074,409.243,172.528,33.615,156.259
C04685=1058.203,221.311,409.218,172.530,33.619,156.260
C04686=1058.208,221.548,409.192,172.532,33.623,156.261
C04687=1058.215,221.785,409.167,172.534,33.627,156.261
C04688=1058.220,222.022,409.141,172.536,33.630,156.262
C04689=1058.226,222.259,409.116,172.538,33.634,156.263
C04690=1058.232,222.496,409.091,172.540,33.638,156.263
C04691=1058.238,222.734,409.066,172.543,33.641,156.264
C04692=1058.244,222.982,409.039,172.545,33.645,156.265
C04693=1058.250,223.231,409.012,172.547,33.649,156.265
C04694=1058.256,223.479,408.986,172.549,33.653,156.266
C04695=1058.262,223.727,408.959,172.551,33.657,156.267
C04696=1058.269,223.976,408.931,172.553,33.660,156.268
C04697=1058.275,224.224,408.905,172.555,33.664,156.268
C04698=1058.281,224.473,408.878,172.557,33.668,156.269
C04699=1058.287,224.722,408.851,172.559,33.672,156.270
C04700=1058.293,224.970,408.825,172.561,33.676,156.271
C04701=1058.300,225.219,408.798,172.563,33.680,156.271
C04702=1058.306,225.467,408.771,172.566,33.683,156.272
C04703=1058.311,225.716,408.745,172.568,33.687,156.273
C04704=1058.318,225.964,408.717,172.570,33.691,156.274
C04705=1058.324,226.212,408.691,172.572,33.695,156.274
C04706=1058.331,226.461,408.664,172.574,33.698,156.275
C04707=1058.337,226.709,408.637,172.576,33.702,156.276
C04708=1058.343,226.959,408.610,172.578,33.706,156.276
C04709=1058.349,227.206,408.583,172.580,33.710,156.277
C04710=1058.355,227.455,408.556,172.582,33.714,156.278
C04711=1058.361,227.704,408.529,172.584,33.717,156.279
C04712=1058.368,227.952,408.503,172.587,33.721,156.279
C04713=1058.374,228.200,408.475,172.589,33.725,156.280
C04714=1058.380,228.449,408.449,172.591,33.729,156.281
C04715=1058.387,228.698,408.422,172.593,33.732,156.281
C04716=1058.392,228.946,408.395,172.595,33.736,156.282
C04717=1058.399,229.194,408.367,172.598,33.740,156.283
C04718=1058.405,229.443,408.340,172.600,33.744,156.284
C04719=1058.411,229.692,408.314,172.602,33.748,156.284
C04720=1058.417,229.940,408.286,172.604,33.751,156.285
C04721=1058.424,230.189,408.259,172.606,33.755,156.286
C04722=1058.430,230.436,408.232,172.609,33.759,156.287
C04723=1058.436,230.685,408.205,172.611,33.763,156.287
C04724=1058.442,230.934,408.178,172.613,33.766,156.288
C04725=1058.449,231.182,408.151,172.615,33.771,156.289
C04726=1058.454,231.431,408.124,172.617,33.774,156.289
C04727=1058.461,231.679,408.096,172.619,33.778,156.290
C04728=1058.467,231.927,408.070,172.621,33.782,156.291
C04729=1058.473,232.176,408.042,172.624,33.786,156.292
C04730=1058.479,232.424,408.015,172.626,33.789,156.292
C04731=1058.485,232.673,407.987,172.629,33.793,156.293
C04732=1058.492,232.922,407.960,172.631,33.797,156.294
C04733=1058.498,233.170,407.933,172.633,33.801,156.295
C04734=1058.504,233.419,407.906,172.635,33.805,156.295
C04735=1058.510,233.667,407.878,172.637,33.808,156.296
C04736=1058.516,233.916,407.851,172.639,33.812,156.297
C04737=1058.522,234.164,407.823,172.641,33.816,156.298
C04738=1058.528,234.412,407.795,172.643,33.820,156.298
C04739=1058.534,234.660,407.769,172.646,33.823,156.299
C04740=1058.540,234.894,407.743,172.649,33.827,156.300
C04741=1058.546,235.127,407.717,172.651,33.831,156.300
C04742=1058.552,235.360,407.691,172.653,33.834,156.301
C04743=1058.558,235.593,407.665,172.655,33.838,156.302
C04744=1058.563,235.827,407.640,172.657,33.842,156.302
C04745=1058.569,236.060,407.614,172.659,33.845,156.303
C04746=1058.575,236.294,407.588,172.661,33.848,156.304
C04747=1058.581,236.527,407.562,172.663,33.852,156.304
C04748=1058.587,236.775,407.535,172.665,33.856,156.305
C04749=1058.593,237.023,407.507,172.668,33.860,156.306
C04750=1058.599,237.271,407.480,172.670,33.863,156.307
C04751=1058.605,237.520,407.452,172.672,33.867,156.307
C04752=1058.612,237.769,407.424,172.674,33.871,156.308
C04753=1058.618,238.016,407.397,172.676,33.875,156.309
C04754=1058.624,238.265,407.370,172.679,33.879,156.310
C04755=1058.630,238.514,407.342,172.681,33.882,156.310
C04756=1058.636,238.762,407.314,172.683,33.886,156.311
C04757=1058.643,239.010,407.286,172.686,33.889,156.312
C04758=1058.650,239.259,407.259,172.688,33.894,156.312
C04759=1058.655,239.507,407.231,172.690,33.897,156.313
C04760=1058.661,239.756,407.204,172.693,33.901,156.314
C04761=1058.668,240.004,407.176,172.695,33.905,156.315
C04762=1058.673,240.252,407.148,172.697,33.908,156.315
C04763=1058.680,240.501,407.120,172.699,33.912,156.316
C04764=1058.687,240.749,407.093,172.701,33.916,156.317
C04765=1058.692,240.997,407.065,172.705,33.920,156.317
C04766=1058.699,241.246,407.037,172.707,33.923,156.318
C04767=1058.705,241.494,407.009,172.709,33.927,156.319
C04768=1058.711,241.743,406.981,172.711,33.931,156.320
C04769=1058.717,241.991,406.954,172.713,33.935,156.320
C04770=1058.723,242.239,406.925,172.715,33.938,156.321
C04771=1058.730,242.488,406.897,172.718,33.942,156.322
C04772=1058.736,242.737,406.869,172.720,33.946,156.322
C04773=1058.742,242.984,406.842,172.723,33.950,156.323
C04774=1058.748,243.233,406.813,172.725,33.954,156.324
C04775=1058.755,243.482,406.786,172.727,33.957,156.325
C04776=1058.760,243.730,406.758,172.730,33.961,156.325
C04777=1058.767,243.978,406.730,172.732,33.965,156.326
C04778=1058.773,244.227,406.702,172.734,33.969,156.327
C04779=1058.779,244.475,406.674,172.736,33.972,156.328
C04780=1058.785,244.723,406.646,172.740,33.976,156.328
C04781=1058.791,244.972,406.618,172.742,33.980,156.329
C04782=1058.798,245.220,406.589,172.744,33.984,156.330
C04783=1058.804,245.469,406.561,172.746,33.987,156.331
C04784=1058.810,245.716,406.534,172.748,33.991,156.331
C04785=1058.816,245.965,406.505,172.751,33.995,156.332
C04786=1058.822,246.214,406.477,172.753,33.999,156.333
C04787=1058.829,246.462,406.448,172.755,34.002,156.334
C04788=1058.834,246.710,406.420,172.758,34.006,156.334
C04789=1058.840,246.958,406.392,172.761,34.010,156.335
C04790=1058.846,247.207,406.364,172.763,34.014,156.336
C04791=1058.853,247.455,406.335,172.765,34.018,156.336
C04792=1058.859,247.704,406.307,172.767,34.021,156.337
C04793=1058.864,247.952,406.279,172.769,34.025,156.338
C04794=1058.870,248.200,406.250,172.772,34.029,156.339
C04795=1058.876,248.449,406.222,172.775,34.033,156.339
C04796=1058.882,248.679,406.196,172.777,34.036,156.340
C04797=1058.888,248.909,406.169,172.779,34.040,156.341
C04798=1058.893,249.139,406.144,172.781,34.044,156.341
C04799=1058.899,249.369,406.117,172.783,34.047,156.342
C04800=1058.904,249.599,406.090,172.785,34.051,156.343
C04801=1058.910,249.830,406.064,172.788,34.054,156.343
C04802=1058.916,250.060,406.038,172.791,34.057,156.344
C04803=1058.922,250.290,406.011,172.793,34.061,156.345
C04804=1058.928,250.538,405.982,172.795,34.065,156.346
C04805=1058.933,250.786,405.954,172.797,34.069,156.346
C04806=1058.939,251.034,405.925,172.800,34.073,156.347
C04807=1058.946,251.283,405.898,172.802,34.076,156.348
C04808=1058.952,251.531,405.869,172.804,34.080,156.349
C04809=1058.958,251.780,405.840,172.807,34.084,156.349
C04810=1058.965,252.028,405.811,172.810,34.088,156.350
C04811=1058.971,252.277,405.783,172.812,34.091,156.351
C04812=1058.977,252.525,405.754,172.814,34.095,156.351
C04813=1058.982,252.773,405.726,172.817,34.099,156.352
C04814=1058.989,253.021,405.697,172.819,34.103,156.353
C04815=1058.995,253.269,405.669,172.821,34.106,156.354
C04816=1059.001,253.518,405.640,172.824,34.110,156.354
C04817=1059.008,253.766,405.611,172.827,34.114,156.355
C04818=1059.014,254.014,405.583,172.829,34.118,156.356
C04819=1059.020,254.263,405.554,172.831,34.121,156.357
C04820=1059.026,254.511,405.525,172.834,34.125,156.357
C04821=1059.033,254.759,405.497,172.836,34.129,156.358
C04822=1059.039,255.007,405.468,172.839,34.133,156.359
C04823=1059.045,255.255,405.439,172.842,34.136,156.360
C04824=1059.051,255.504,405.411,172.844,34.140,156.360
C04825=1059.057,255.752,405.381,172.846,34.144,156.361
C04826=1059.064,256.000,405.352,172.849,34.147,156.362
C04827=1059.070,256.249,405.324,172.851,34.151,156.363
C04828=1059.076,256.497,405.295,172.853,34.155,156.363
C04829=1059.082,256.745,405.266,172.857,34.159,156.364
C04830=1059.088,256.994,405.237,172.859,34.162,156.365
C04831=1059.095,257.242,405.209,172.861,34.166,156.365
C04832=1059.101,257.490,405.180,172.864,34.170,156.366
C04833=1059.108,257.738,405.151,172.866,34.174,156.367
C04834=1059.114,257.986,405.122,172.869,34.177,156.368
C04835=1059.120,258.235,405.093,172.872,34.181,156.368
C04836=1059.126,258.483,405.064,172.874,34.185,156.369
C04837=1059.132,258.731,405.036,172.877,34.188,156.370
C04838=1059.138,258.980,405.007,172.879,34.192,156.370
C04839=1059.145,259.228,404.978,172.881,34.196,156.371
C04840=1059.151,259.476,404.949,172.884,34.200,156.372
C04841=1059.158,259.725,404.919,172.887,34.203,156.373
C04842=1059.164,259.973,404.890,172.890,34.207,156.373
C04843=1059.170,260.221,404.861,172.892,34.211,156.374
C04844=1059.177,260.469,404.832,172.894,34.214,156.375
C04845=1059.184,260.717,404.804,172.897,34.218,156.376
C04846=1059.190,260.965,404.775,172.899,34.222,156.376
C04847=1059.196,261.213,404.746,172.903,34.226,156.377
C04848=1059.203,261.462,404.716,172.905,34.229,156.378
C04849=1059.209,261.710,404.687,172.907,34.233,156.378
C04850=1059.215,261.958,404.658,172.910,34.236,156.379
C04851=1059.222,262.206,404.629,172.912,34.240,156.380
C04852=1059.228,262.436,404.602,172.914,34.244,156.381
C04853=1059.233,262.665,404.576,172.918,34.247,156.381
C04854=1059.240,262.894,404.548,172.920,34.250,156.382
C04855=1059.245,263.123,404.521,172.922,34.254,156.383
C04856=1059.251,263.353,404.495,172.924,34.257,156.383
C04857=1059.256,263.582,404.467,172.927,34.261,156.384
C04858=1059.262,263.810,404.440,172.929,34.264,156.385
C04859=1059.268,264.040,404.413,172.931,34.268,156.385
C04860=1059.274,264.288,404.384,172.935,34.271,156.386
C04861=1059.280,264.536,404.354,172.937,34.275,156.387
C04862=1059.286,264.784,404.325,172.939,34.279,156.388
C04863=1059.293,265.032,404.296,172.942,34.283,156.388
C04864=1059.299,265.281,404.266,172.944,34.287,156.389
C04865=1059.305,265.529,404.236,172.948,34.291,156.390
C04866=1059.311,265.777,404.207,172.950,34.294,156.391
C04867=1059.317,266.025,404.177,172.953,34.298,156.391
C04868=1059.324,266.273,404.148,172.955,34.302,156.392
C04869=1059.330,266.521,404.119,172.957,34.305,156.393
C04870=1059.336,266.770,404.089,172.960,34.309,156.393
C04871=1059.342,267.018,404.060,172.963,34.313,156.394
C04872=1059.349,267.266,404.030,172.966,34.317,156.395
C04873=1059.354,267.514,404.000,172.968,34.320,156.396
C04874=1059.361,267.763,403.970,172.971,34.324,156.396
C04875=1059.368,268.011,403.941,172.973,34.328,156.397
C04876=1059.373,268.259,403.911,172.977,34.332,156.398
C04877=1059.380,268.507,403.882,172.979,34.336,156.399
C04878=1059.387,268.756,403.852,172.982,34.339,156.399
C04879=1059.392,269.003,403.822,172.984,34.343,156.400
C04880=1059.399,269.251,403.793,172.987,34.347,156.401
C04881=1059.404,269.499,403.762,172.989,34.351,156.402
C04882=1059.411,269.748,403.733,172.993,34.355,156.403
C04883=1059.417,269.996,403.703,172.995,34.358,156.403
C04884=1059.423,270.244,403.674,172.997,34.362,156.404
C04885=1059.429,270.492,403.643,173.000,34.366,156.405
C04886=1059.436,270.741,403.614,173.002,34.370,156.405
C04887=1059.442,270.989,403.584,173.006,34.373,156.406
C04888=1059.448,271.237,403.555,173.008,34.377,156.407
C04889=1059.454,271.484,403.524,173.011,34.381,156.408
C04890=1059.461,271.733,403.494,173.013,34.385,156.408
C04891=1059.467,271.981,403.464,173.016,34.388,156.409
C04892=1059.473,272.229,403.435,173.020,34.392,156.410
C04893=1059.480,272.477,403.404,173.022,34.396,156.411
C04894=1059.486,272.725,403.375,173.025,34.400,156.411
C04895=1059.492,272.973,403.345,173.027,34.404,156.412
C04896=1059.499,273.221,403.314,173.030,34.407,156.413
C04897=1059.504,273.470,403.285,173.032,34.411,156.414
C04898=1059.510,273.718,403.254,173.036,34.415,156.415
C04899=1059.517,273.966,403.224,173.038,34.419,156.415
C04900=1059.523,274.214,403.194,173.041,34.423,156.416
C04901=1059.529,274.462,403.165,173.043,34.427,156.417
C04902=1059.536,274.710,403.134,173.046,34.430,156.418
C04903=1059.542,274.958,403.104,173.049,34.434,156.418
C04904=1059.549,275.206,403.074,173.052,34.438,156.419
C04905=1059.555,275.454,403.043,173.054,34.441,156.420
C04906=1059.560,275.702,403.013,173.057,34.446,156.421
C04907=1059.567,275.951,402.984,173.059,34.449,156.421
C04908=1059.572,276.182,402.955,173.063,34.453,156.422
C04909=1059.578,276.413,402.927,173.065,34.456,156.423
C04910=1059.584,276.644,402.899,173.068,34.460,156.423
C04911=1059.590,276.875,402.871,173.070,34.464,156.424
C04912=1059.595,277.106,402.842,173.072,34.467,156.425
C04913=1059.601,277.337,402.814,173.076,34.471,156.426
C04914=1059.607,277.568,402.786,173.078,34.474,156.426
C04915=1059.613,277.799,402.758,173.081,34.478,156.427
C04916=1059.619,278.047,402.727,173.083,34.482,156.428
C04917=1059.625,278.296,402.697,173.086,34.486,156.429
C04918=1059.632,278.543,402.667,173.089,34.489,156.429
C04919=1059.638,278.792,402.636,173.092,34.493,156.430
C04920=1059.644,279.039,402.606,173.094,34.497,156.431
C04921=1059.651,279.288,402.575,173.097,34.501,156.432
C04922=1059.657,279.535,402.545,173.101,34.505,156.432
C04923=1059.664,279.783,402.514,173.103,34.508,156.433
C04924=1059.670,280.031,402.484,173.106,34.512,156.434
C04925=1059.676,280.280,402.453,173.108,34.516,156.435
C04926=1059.682,280.527,402.422,173.111,34.520,156.435
C04927=1059.688,280.776,402.392,173.115,34.524,156.436
C04928=1059.694,281.024,402.361,173.117,34.527,156.437
C04929=1059.700,281.272,402.331,173.120,34.532,156.438
C04930=1059.707,281.520,402.300,173.122,34.535,156.439
C04931=1059.713,281.767,402.269,173.125,34.539,156.439
C04932=1059.719,282.016,402.239,173.129,34.543,156.440
C04933=1059.725,282.264,402.208,173.131,34.547,156.441
C04934=1059.732,282.512,402.177,173.134,34.551,156.442
C04935=1059.737,282.759,402.146,173.136,34.555,156.442
C04936=1059.744,283.008,402.116,173.140,34.558,156.443
C04937=1059.751,283.256,402.084,173.143,34.563,156.444
C04938=1059.756,283.504,402.054,173.145,34.566,156.445
C04939=1059.763,283.752,402.023,173.148,34.570,156.446
C04940=1059.769,283.999,401.992,173.151,34.574,156.446
C04941=1059.775,284.248,401.961,173.154,34.578,156.447
C04942=1059.781,284.496,401.931,173.157,34.582,156.448
C04943=1059.788,284.744,401.900,173.160,34.586,156.449
C04944=1059.794,284.991,401.869,173.162,34.589,156.449
C04945=1059.800,285.239,401.838,173.166,34.594,156.450
C04946=1059.807,285.488,401.807,173.169,34.597,156.451
C04947=1059.813,285.736,401.777,173.171,34.601,156.452
C04948=1059.819,285.984,401.745,173.174,34.605,156.453
C04949=1059.826,286.232,401.715,173.177,34.609,156.453
C04950=1059.832,286.479,401.684,173.180,34.613,156.454
C04951=1059.838,286.728,401.653,173.183,34.617,156.455
C04952=1059.844,286.975,401.622,173.186,34.620,156.456
C04953=1059.851,287.224,401.591,173.188,34.624,156.457
C04954=1059.858,287.472,401.560,173.192,34.628,156.457
C04955=1059.864,287.719,401.529,173.195,34.632,156.458
C04956=1059.870,287.967,401.498,173.197,34.636,156.459
C04957=1059.877,288.215,401.466,173.200,34.640,156.460
C04958=1059.883,288.464,401.436,173.204,34.644,156.460
C04959=1059.889,288.711,401.404,173.206,34.648,156.461
C04960=1059.895,288.959,401.373,173.209,34.651,156.462
C04961=1059.901,289.207,401.342,173.212,34.655,156.463
C04962=1059.908,289.455,401.311,173.215,34.659,156.464
C04963=1059.915,289.703,401.279,173.218,34.663,156.464
C04964=1059.921,289.939,401.249,173.221,34.667,156.465
C04965=1059.926,290.176,401.220,173.223,34.671,156.466
C04966=1059.932,290.412,401.190,173.226,34.674,156.467
C04967=1059.938,290.648,401.160,173.230,34.678,156.467
C04968=1059.944,290.885,401.130,173.232,34.682,156.468
C04969=1059.951,291.121,401.100,173.235,34.686,156.469
C04970=1059.957,291.358,401.070,173.237,34.689,156.470
C04971=1059.963,291.595,401.041,173.241,34.693,156.470
C04972=1059.968,291.842,401.009,173.244,34.697,156.471
C04973=1059.975,292.090,400.978,173.246,34.701,156.472
C04974=1059.981,292.338,400.946,173.249,34.705,156.473
C04975=1059.987,292.587,400.914,173.253,34.709,156.474
C04976=1059.993,292.834,400.883,173.256,34.713,156.474
C04977=1060.000,293.082,400.852,173.258,34.717,156.475
C04978=1060.006,293.330,400.820,173.261,34.721,156.476
C04979=1060.013,293.578,400.788,173.265,34.725,156.477
C04980=1060.019,293.825,400.757,173.268,34.729,156.478
C04981=1060.025,294.073,400.725,173.270,34.732,156.478
C04982=1060.032,294.321,400.694,173.273,34.737,156.479
C04983=1060.038,294.569,400.662,173.277,34.741,156.480
C04984=1060.044,294.817,400.630,173.280,34.744,156.481
C04985=1060.051,295.065,400.599,173.282,34.748,156.482
C04986=1060.057,295.313,400.567,173.285,34.753,156.483
C04987=1060.063,295.560,400.536,173.289,34.756,156.483
C04988=1060.069,295.809,400.504,173.292,34.760,156.484
C04989=1060.076,296.057,400.472,173.295,34.764,156.485
C04990=1060.082,296.305,400.440,173.297,34.769,156.486
C04991=1060.089,296.553,400.409,173.301,34.772,156.487
C04992=1060.095,296.800,400.378,173.304,34.776,156.487
C04993=1060.101,297.048,400.345,173.307,34.780,156.488
C04994=1060.107,297.296,400.313,173.311,34.785,156.489
C04995=1060.113,297.544,400.281,173.313,34.789,156.490
C04996=1060.120,297.792,400.250,173.316,34.793,156.491
C04997=1060.126,298.039,400.217,173.319,34.797,156.492
C04998=1060.131,298.287,400.185,173.323,34.800,156.492
C04999=1060.137,298.535,400.153,173.325,34.805,156.493
C05000=1060.145,298.782,400.121,173.328,34.809,156.494
C05001=1060.150,299.031,400.089,173.331,34.813,156.495
C05002=1060.156,299.279,400.057,173.335,34.817,156.496
C05003=1060.162,299.526,400.025,173.338,34.821,156.497
C05004=1060.169,299.774,399.993,173.340,34.825,156.497
C05005=1060.175,300.022,399.961,173.344,34.829,156.498
C05006=1060.181,300.269,399.928,173.347,34.833,156.499
C05007=1060.187,300.518,399.896,173.350,34.838,156.500
C05008=1060.194,300.765,399.864,173.353,34.842,156.501
C05009=1060.200,301.013,399.832,173.357,34.846,156.502
C05010=1060.206,301.261,399.799,173.359,34.849,156.502
C05011=1060.212,301.509,399.767,173.362,34.853,156.503
C05012=1060.219,301.757,399.735,173.366,34.858,156.504
C05013=1060.225,302.004,399.704,173.369,34.862,156.505
C05014=1060.231,302.251,399.671,173.372,34.866,156.506
C05015=1060.237,302.500,399.639,173.375,34.870,156.507
C05016=1060.243,302.747,399.606,173.379,34.874,156.508
C05017=1060.249,302.995,399.574,173.381,34.878,156.508
C05018=1060.256,303.243,399.542,173.384,34.882,156.509
C05019=1060.262,303.491,399.510,173.388,34.886,156.510
C05020=1060.268,303.735,399.477,173.391,34.891,156.511
C05021=1060.275,303.979,399.445,173.394,34.895,156.512
C05022=1060.281,304.224,399.413,173.397,34.899,156.513
C05023=1060.288,304.467,399.381,173.401,34.902,156.513
C05024=1060.294,304.711,399.350,173.403,34.906,156.514
C05025=1060.300,304.955,399.318,173.406,34.911,156.515
C05026=1060.307,305.199,399.286,173.410,34.915,156.516
C05027=1060.312,305.444,399.254,173.413,34.919,156.517
C05028=1060.319,305.692,399.221,173.416,34.923,156.518
C05029=1060.325,305.939,399.188,173.419,34.927,156.518
C05030=1060.331,306.187,399.156,173.423,34.931,156.519
C05031=1060.338,306.435,399.124,173.426,34.935,156.520
C05032=1060.344,306.682,399.091,173.429,34.939,156.521
C05033=1060.351,306.931,399.058,173.432,34.943,156.522
C05034=1060.358,307.178,399.026,173.435,34.948,156.523
C05035=1060.364,307.426,398.993,173.438,34.952,156.524
C05036=1060.370,307.674,398.961,173.442,34.956,156.524
C05037=1060.376,307.922,398.928,173.445,34.960,156.525
C05038=1060.383,308.169,398.896,173.448,34.964,156.526
C05039=1060.389,308.416,398.863,173.451,34.968,156.527
C05040=1060.396,308.665,398.830,173.455,34.972,156.528
C05041=1060.403,308.912,398.797,173.458,34.976,156.529
C05042=1060.409,309.160,398.765,173.461,34.980,156.530
C05043=1060.415,309.408,398.732,173.465,34.985,156.530
C05044=1060.422,309.655,398.699,173.468,34.989,156.531
C05045=1060.428,309.903,398.666,173.471,34.993,156.532
C05046=1060.435,310.151,398.633,173.475,34.997,156.533
C05047=1060.441,310.399,398.600,173.478,35.001,156.534
C05048=1060.448,310.646,398.568,173.481,35.005,156.535
C05049=1060.455,310.894,398.535,173.485,35.009,156.536
C05050=1060.461,311.142,398.502,173.488,35.013,156.536
C05051=1060.468,311.389,398.470,173.491,35.018,156.537
C05052=1060.474,311.637,398.437,173.495,35.022,156.538
C05053=1060.481,311.885,398.404,173.498,35.026,156.539
C05054=1060.487,312.132,398.370,173.501,35.030,156.540
C05055=1060.494,312.380,398.338,173.504,35.034,156.541
C05056=1060.500,312.628,398.305,173.508,35.038,156.542
C05057=1060.507,312.876,398.272,173.511,35.043,156.543
C05058=1060.513,313.123,398.239,173.514,35.047,156.543
C05059=1060.520,313.372,398.206,173.518,35.051,156.544
C05060=1060.527,313.619,398.173,173.521,35.055,156.545
C05061=1060.533,313.866,398.140,173.524,35.059,156.546
C05062=1060.540,314.114,398.107,173.528,35.064,156.547
C05063=1060.546,314.362,398.073,173.531,35.068,156.548
C05064=1060.552,314.609,398.040,173.534,35.072,156.549
C05065=1060.557,314.857,398.007,173.538,35.076,156.550
C05066=1060.565,315.105,397.973,173.541,35.081,156.551
C05067=1060.570,315.353,397.939,173.544,35.085,156.552
C05068=1060.577,315.600,397.906,173.548,35.090,156.553
C05069=1060.583,315.848,397.872,173.551,35.094,156.553
C05070=1060.590,316.095,397.839,173.554,35.099,156.554
C05071=1060.595,316.343,397.805,173.558,35.103,156.555
C05072=1060.602,316.591,397.772,173.561,35.107,156.556
C05073=1060.609,316.839,397.739,173.564,35.111,156.557
C05074=1060.614,317.086,397.705,173.568,35.115,156.558
C05075=1060.621,317.334,397.672,173.571,35.120,156.559
C05076=1060.628,317.580,397.638,173.575,35.124,156.560
C05077=1060.634,317.826,397.605,173.578,35.129,156.561
C05078=1060.640,318.072,397.572,173.581,35.133,156.562
C05079=1060.646,318.318,397.538,173.585,35.138,156.563
C05080=1060.652,318.564,397.505,173.588,35.142,156.563
C05081=1060.659,318.810,397.471,173.591,35.146,156.564
C05082=1060.665,319.057,397.438,173.595,35.150,156.565
C05083=1060.671,319.302,397.404,173.598,35.154,156.566
C05084=1060.678,319.549,397.370,173.601,35.159,156.567
C05085=1060.684,319.798,397.337,173.605,35.163,156.568
C05086=1060.691,320.045,397.303,173.609,35.168,156.569
C05087=1060.697,320.293,397.269,173.612,35.173,156.570
C05088=1060.703,320.540,397.236,173.616,35.177,156.571
C05089=1060.710,320.788,397.202,173.619,35.181,156.572
C05090=1060.716,321.035,397.168,173.623,35.185,156.573
C05091=1060.723,321.283,397.134,173.626,35.190,156.574
C05092=1060.729,321.530,397.100,173.629,35.194,156.575
C05093=1060.736,321.778,397.066,173.633,35.199,156.576
C05094=1060.741,322.026,397.032,173.636,35.203,156.577
C05095=1060.749,322.274,396.999,173.639,35.207,156.577
C05096=1060.755,322.521,396.965,173.644,35.212,156.578
C05097=1060.762,322.769,396.931,173.647,35.216,156.579
C05098=1060.768,323.017,396.896,173.651,35.221,156.580
C05099=1060.775,323.264,396.863,173.654,35.225,156.581
C05100=1060.781,323.512,396.828,173.657,35.229,156.582
C05101=1060.787,323.759,396.794,173.661,35.234,156.583
C05102=1060.794,324.007,396.761,173.664,35.238,156.584
C05103=1060.801,324.255,396.726,173.668,35.243,156.585
C05104=1060.807,324.502,396.693,173.672,35.247,156.586
C05105=1060.814,324.750,396.658,173.675,35.251,156.587
C05106=1060.820,324.998,396.624,173.679,35.256,156.588
C05107=1060.827,325.245,396.590,173.682,35.261,156.589
C05108=1060.833,325.493,396.556,173.685,35.265,156.590
C05109=1060.841,325.740,396.522,173.690,35.269,156.591
C05110=1060.846,325.988,396.488,173.693,35.274,156.592
C05111=1060.853,326.236,396.454,173.696,35.279,156.593
C05112=1060.860,326.483,396.419,173.700,35.283,156.594
C05113=1060.866,326.730,396.385,173.703,35.287,156.595
C05114=1060.873,326.978,396.351,173.707,35.292,156.596
C05115=1060.880,327.226,396.317,173.711,35.296,156.596
C05116=1060.886,327.474,396.282,173.714,35.301,156.597
C05117=1060.893,327.720,396.248,173.718,35.305,156.598
C05118=1060.900,327.968,396.214,173.721,35.310,156.599
C05119=1060.906,328.216,396.179,173.726,35.314,156.600
C05120=1060.913,328.464,396.146,173.729,35.319,156.601
C05121=1060.920,328.711,396.110,173.732,35.323,156.602
C05122=1060.926,328.958,396.076,173.736,35.328,156.603
C05123=1060.933,329.206,396.043,173.739,35.332,156.604
C05124=1060.940,329.453,396.007,173.744,35.337,156.605
C05125=1060.946,329.701,395.973,173.747,35.341,156.606
C05126=1060.954,329.949,395.939,173.750,35.346,156.607
C05127=1060.960,330.196,395.904,173.754,35.350,156.608
C05128=1060.967,330.444,395.870,173.758,35.355,156.609
C05129=1060.973,330.691,395.835,173.762,35.360,156.610
C05130=1060.980,330.939,395.800,173.765,35.364,156.611
C05131=1060.986,331.186,395.765,173.769,35.369,156.612
C05132=1060.993,331.429,395.731,173.773,35.373,156.613
C05133=1061.000,331.673,395.698,173.776,35.378,156.614
C05134=1061.005,331.916,395.663,173.780,35.383,156.615
C05135=1061.012,332.159,395.629,173.783,35.387,156.616
C05136=1061.018,332.402,395.595,173.787,35.392,156.617
C05137=1061.025,332.645,395.560,173.791,35.397,156.618
C05138=1061.032,332.888,395.526,173.795,35.401,156.619
C05139=1061.038,333.132,395.492,173.798,35.406,156.620
C05140=1061.044,333.380,395.457,173.801,35.410,156.621
C05141=1061.051,333.627,395.422,173.806,35.415,156.622
C05142=1061.058,333.874,395.387,173.809,35.420,156.623
C05143=1061.064,334.122,395.353,173.813,35.424,156.624
C05144=1061.071,334.369,395.318,173.816,35.429,156.625
C05145=1061.077,334.616,395.282,173.821,35.434,156.626
C05146=1061.084,334.864,395.247,173.824,35.438,156.627
C05147=1061.091,335.111,395.212,173.827,35.443,156.628
C05148=1061.097,335.359,395.178,173.832,35.448,156.629
C05149=1061.103,335.607,395.142,173.835,35.452,156.630
C05150=1061.110,335.854,395.107,173.839,35.457,156.631
C05151=1061.117,336.102,395.072,173.843,35.462,156.632
C05152=1061.124,336.349,395.037,173.847,35.467,156.633
C05153=1061.130,336.596,395.002,173.850,35.471,156.634
C05154=1061.137,336.844,394.966,173.855,35.476,156.635
C05155=1061.144,337.091,394.931,173.858,35.481,156.636
C05156=1061.150,337.339,394.896,173.861,35.486,156.637
C05157=1061.157,337.586,394.860,173.866,35.491,156.639
C05158=1061.163,337.833,394.825,173.869,35.495,156.640
C05159=1061.170,338.081,394.790,173.873,35.500,156.641
C05160=1061.176,338.329,394.754,173.877,35.505,156.642
C05161=1061.183,338.576,394.719,173.881,35.510,156.643
C05162=1061.190,338.823,394.684,173.884,35.515,156.644
C05163=1061.196,339.071,394.648,173.889,35.520,156.645
C05164=1061.203,339.318,394.613,173.892,35.525,156.646
C05165=1061.210,339.565,394.577,173.897,35.530,156.647
C05166=1061.216,339.813,394.542,173.900,35.534,156.648
C05167=1061.223,340.061,394.506,173.904,35.539,156.649
C05168=1061.230,340.308,394.471,173.908,35.544,156.650
C05169=1061.236,340.555,394.435,173.912,35.549,156.651
C05170=1061.243,340.803,394.399,173.915,35.554,156.652
C05171=1061.250,341.050,394.364,173.920,35.559,156.654
C05172=1061.256,341.297,394.328,173.923,35.563,156.655
C05173=1061.263,341.544,394.293,173.928,35.569,156.656
C05174=1061.269,341.792,394.257,173.931,35.574,156.657
C05175=1061.277,342.039,394.221,173.936,35.578,156.658
C05176=1061.283,342.287,394.186,173.939,35.583,156.659
C05177=1061.289,342.535,394.150,173.943,35.588,156.660
C05178=1061.296,342.781,394.114,173.947,35.593,156.661
C05179=1061.303,343.029,394.079,173.951,35.598,156.662
C05180=1061.310,343.276,394.042,173.955,35.603,156.663
C05181=1061.317,343.524,394.007,173.959,35.608,156.664
C05182=1061.323,343.771,393.971,173.963,35.613,156.665
C05183=1061.330,344.018,393.935,173.967,35.618,156.667
C05184=1061.336,344.265,393.899,173.970,35.623,156.668
C05185=1061.343,344.514,393.863,173.975,35.628,156.669
C05186=1061.350,344.760,393.827,173.978,35.633,156.670
C05187=1061.356,345.007,393.791,173.983,35.638,156.671
C05188=1061.363,345.248,393.756,173.986,35.643,156.672
C05189=1061.370,345.489,393.720,173.991,35.648,156.673
C05190=1061.376,345.730,393.685,173.994,35.653,156.674
C05191=1061.383,345.971,393.650,173.998,35.658,156.675
C05192=1061.389,346.211,393.615,174.002,35.663,156.676
C05193=1061.396,346.453,393.579,174.006,35.668,156.678
C05194=1061.402,346.694,393.544,174.010,35.673,156.679
C05195=1061.409,346.934,393.509,174.014,35.678,156.680
C05196=1061.415,347.181,393.473,174.017,35.683,156.681
C05197=1061.422,347.430,393.438,174.022,35.688,156.682
C05198=1061.429,347.677,393.401,174.025,35.693,156.683
C05199=1061.435,347.924,393.365,174.030,35.699,156.684
C05200=1061.443,348.171,393.328,174.035,35.704,156.686
C05201=1061.449,348.418,393.292,174.038,35.709,156.687
C05202=1061.455,348.665,393.256,174.043,35.714,156.688
C05203=1061.462,348.913,393.219,174.046,35.719,156.689
C05204=1061.469,349.160,393.183,174.051,35.724,156.690
C05205=1061.476,349.407,393.146,174.054,35.729,156.691
C05206=1061.483,349.655,393.110,174.059,35.734,156.692
C05207=1061.490,349.901,393.074,174.062,35.740,156.694
C05208=1061.497,350.149,393.037,174.067,35.745,156.695
C05209=1061.503,350.396,393.001,174.071,35.750,156.696
C05210=1061.510,350.644,392.964,174.075,35.755,156.697
C05211=1061.517,350.891,392.928,174.080,35.760,156.698
C05212=1061.524,351.138,392.891,174.083,35.766,156.700
C05213=1061.530,351.385,392.855,174.088,35.771,156.701
C05214=1061.538,351.633,392.817,174.091,35.776,156.702
C05215=1061.544,351.880,392.781,174.096,35.781,156.703
C05216=1061.551,352.127,392.744,174.100,35.787,156.704
C05217=1061.557,352.374,392.707,174.104,35.792,156.705
C05218=1061.564,352.621,392.672,174.109,35.798,156.707
C05219=1061.572,352.868,392.634,174.112,35.803,156.708
C05220=1061.578,353.115,392.598,174.117,35.808,156.709
C05221=1061.585,353.363,392.561,174.120,35.814,156.710
C05222=1061.591,353.610,392.524,174.125,35.819,156.711
C05223=1061.598,353.857,392.487,174.130,35.824,156.713
C05224=1061.606,354.104,392.449,174.133,35.829,156.714
C05225=1061.612,354.351,392.413,174.138,35.835,156.715
C05226=1061.619,354.599,392.376,174.142,35.840,156.716
C05227=1061.626,354.846,392.339,174.146,35.846,156.718
C05228=1061.632,355.093,392.302,174.151,35.851,156.719
C05229=1061.639,355.340,392.265,174.154,35.857,156.720
C05230=1061.646,355.588,392.228,174.159,35.862,156.721
C05231=1061.653,355.835,392.191,174.163,35.867,156.722
C05232=1061.660,356.081,392.153,174.167,35.873,156.724
C05233=1061.667,356.329,392.117,174.172,35.879,156.725
C05234=1061.674,356.575,392.079,174.176,35.884,156.726
C05235=1061.680,356.823,392.043,174.180,35.889,156.727
C05236=1061.688,357.070,392.005,174.185,35.895,156.729
C05237=1061.694,357.317,391.968,174.189,35.900,156.730
C05238=1061.701,357.565,391.930,174.193,35.906,156.731
C05239=1061.708,357.812,391.893,174.197,35.911,156.732
C05240=1061.714,358.058,391.856,174.202,35.917,156.734
C05241=1061.722,358.305,391.818,174.207,35.922,156.735
C05242=1061.729,358.553,391.781,174.210,35.928,156.736
C05243=1061.736,358.800,391.744,174.215,35.933,156.737
C05244=1061.742,359.043,391.707,174.220,35.939,156.739
C05245=1061.750,359.286,391.670,174.223,35.944,156.740
C05246=1061.756,359.529,391.633,174.228,35.950,156.741
C05247=1061.763,359.772,391.596,174.233,35.955,156.742
C05248=1061.770,360.015,391.560,174.236,35.961,156.744
C05249=1061.776,360.258,391.523,174.241,35.966,156.745
C05250=1061.783,360.501,391.486,174.246,35.972,156.746
C05251=1061.790,360.744,391.449,174.249,35.978,156.747
C05252=1061.797,360.991,391.411,174.254,35.983,156.749
C05253=1061.804,361.239,391.373,174.259,35.989,156.750
C05254=1061.810,361.485,391.336,174.263,35.994,156.751
C05255=1061.818,361.732,391.299,174.267,36.000,156.753
C05256=1061.824,361.980,391.261,174.272,36.006,156.754
C05257=1061.832,362.226,391.222,174.276,36.012,156.755
C05258=1061.839,362.473,391.185,174.281,36.017,156.757
C05259=1061.845,362.720,391.147,174.285,36.023,156.758
C05260=1061.852,362.967,391.110,174.289,36.029,156.759
C05261=1061.859,363.214,391.072,174.294,36.034,156.760
C05262=1061.867,363.461,391.034,174.299,36.040,156.762
C05263=1061.873,363.708,390.996,174.303,36.046,156.763
C05264=1061.881,363.955,390.958,174.307,36.052,156.764
C05265=1061.887,364.203,390.920,174.312,36.058,156.766
C05266=1061.895,364.449,390.882,174.317,36.063,156.767
C05267=1061.901,364.697,390.844,174.321,36.069,156.769
C05268=1061.908,364.943,390.806,174.326,36.075,156.770
C05269=1061.915,365.190,390.768,174.330,36.081,156.771
C05270=1061.922,365.437,390.730,174.334,36.087,156.773
C05271=1061.929,365.684,390.691,174.339,36.093,156.774
C05272=1061.936,365.931,390.654,174.344,36.098,156.775
C05273=1061.943,366.178,390.615,174.349,36.105,156.777
C05274=1061.949,366.425,390.577,174.353,36.110,156.778
C05275=1061.957,366.672,390.539,174.357,36.116,156.779
C05276=1061.964,366.919,390.500,174.362,36.122,156.781
C05277=1061.971,367.166,390.462,174.367,36.128,156.782
C05278=1061.978,367.413,390.423,174.371,36.134,156.784
C05279=1061.985,367.659,390.385,174.376,36.140,156.785
C05280=1061.992,367.907,390.347,174.381,36.146,156.786
C05281=1061.999,368.153,390.308,174.386,36.152,156.788
C05282=1062.006,368.400,390.270,174.390,36.158,156.789
C05283=1062.013,368.647,390.232,174.394,36.164,156.791
C05284=1062.020,368.894,390.194,174.399,36.170,156.792
C05285=1062.027,369.141,390.155,174.404,36.176,156.793
C05286=1062.034,369.388,390.116,174.408,36.182,156.795
C05287=1062.041,369.634,390.078,174.413,36.188,156.796
C05288=1062.048,369.882,390.040,174.418,36.194,156.798
C05289=1062.055,370.129,390.000,174.423,36.200,156.799
C05290=1062.063,370.376,389.962,174.428,36.207,156.800
C05291=1062.070,370.622,389.923,174.432,36.213,156.802
C05292=1062.076,370.869,389.884,174.437,36.219,156.803
C05293=1062.084,371.116,389.846,174.442,36.225,156.805
C05294=1062.091,371.363,389.807,174.447,36.231,156.806
C05295=1062.099,371.610,389.769,174.451,36.237,156.808
C05296=1062.106,371.857,389.730,174.456,36.243,156.809
C05297=1062.113,372.103,389.691,174.461,36.249,156.810
C05298=1062.119,372.350,389.652,174.466,36.255,156.812
C05299=1062.128,372.597,389.614,174.471,36.262,156.813
C05300=1062.135,372.854,389.573,174.476,36.268,156.815
C05301=1062.142,373.111,389.532,174.480,36.275,156.816
C05302=1062.149,373.368,389.492,174.485,36.282,156.818
C05303=1062.157,373.626,389.451,174.490,36.288,156.820
C05304=1062.164,373.872,389.411,174.495,36.294,156.821
C05305=1062.171,374.119,389.373,174.500,36.301,156.823
C05306=1062.177,374.366,389.334,174.505,36.307,156.824
C05307=1062.185,374.613,389.294,174.510,36.313,156.825
C05308=1062.192,374.859,389.255,174.514,36.320,156.827
C05309=1062.199,375.106,389.215,174.519,36.326,156.829
C05310=1062.206,375.352,389.177,174.524,36.332,156.830
C05311=1062.213,375.600,389.137,174.529,36.339,156.832
C05312=1062.220,375.846,389.098,174.534,36.345,156.833
C05313=1062.227,376.093,389.059,174.539,36.352,156.835
C05314=1062.235,376.340,389.019,174.545,36.358,156.836
C05315=1062.242,376.587,388.980,174.549,36.365,156.838
C05316=1062.249,376.833,388.941,174.554,36.371,156.839
C05317=1062.257,377.080,388.901,174.559,36.378,156.841
C05318=1062.263,377.327,388.862,174.564,36.384,156.842
C05319=1062.271,377.574,388.822,174.569,36.390,156.844
C05320=1062.278,377.820,388.782,174.574,36.397,156.845
C05321=1062.285,378.067,388.744,174.579,36.404,156.847
C05322=1062.293,378.314,388.704,174.584,36.410,156.848
C05323=1062.300,378.560,388.664,174.589,36.416,156.850
C05324=1062.307,378.807,388.625,174.593,36.423,156.851
C05325=1062.314,379.053,388.585,174.599,36.430,156.853
C05326=1062.322,379.300,388.545,174.604,36.436,156.855
C05327=1062.329,379.547,388.506,174.609,36.443,156.856
C05328=1062.337,379.793,388.466,174.614,36.449,156.858
C05329=1062.344,380.040,388.426,174.619,36.456,156.859
C05330=1062.352,380.287,388.387,174.624,36.463,156.861
C05331=1062.359,380.533,388.348,174.629,36.469,156.862
C05332=1062.366,380.780,388.308,174.635,36.476,156.864
C05333=1062.374,381.027,388.268,174.640,36.483,156.866
C05334=1062.380,381.274,388.228,174.645,36.490,156.867
C05335=1062.388,381.520,388.187,174.650,36.496,156.869
C05336=1062.396,381.766,388.147,174.655,36.503,156.871
C05337=1062.403,382.013,388.107,174.660,36.510,156.872
C05338=1062.410,382.260,388.067,174.666,36.517,156.874
C05339=1062.417,382.507,388.028,174.671,36.524,156.875
C05340=1062.424,382.753,387.987,174.676,36.530,156.877
C05341=1062.432,382.999,387.947,174.681,36.537,156.879
C05342=1062.439,383.246,387.907,174.686,36.544,156.880
C05343=1062.446,383.493,387.867,174.692,36.551,156.882
C05344=1062.454,383.739,387.826,174.697,36.558,156.884
C05345=1062.460,383.986,387.786,174.702,36.565,156.885
C05346=1062.468,384.232,387.746,174.707,36.572,156.887
C05347=1062.476,384.479,387.705,174.713,36.579,156.889
C05348=1062.482,384.725,387.665,174.718,36.586,156.890
C05349=1062.490,384.972,387.625,174.723,36.593,156.892
C05350=1062.497,385.219,387.584,174.728,36.600,156.894
C05351=1062.505,385.466,387.544,174.734,36.606,156.895
C05352=1062.513,385.711,387.504,174.739,36.614,156.897
C05353=1062.520,385.958,387.463,174.744,36.621,156.899
C05354=1062.528,386.205,387.423,174.750,36.628,156.901
C05355=1062.535,386.451,387.381,174.755,36.635,156.902
C05356=1062.543,386.733,387.335,174.761,36.643,156.904
C05357=1062.551,387.014,387.289,174.767,36.651,156.906
C05358=1062.560,387.295,387.243,174.773,36.659,156.908
C05359=1062.569,387.576,387.196,174.780,36.667,156.910
C05360=1062.577,387.830,387.155,174.785,36.674,156.912
C05361=1062.584,388.082,387.113,174.791,36.682,156.914
C05362=1062.592,388.336,387.072,174.796,36.689,156.915
C05363=1062.600,388.588,387.029,174.802,36.697,156.917
C05364=1062.608,388.835,386.990,174.807,36.704,156.919
C05365=1062.615,389.082,386.948,174.812,36.711,156.921
C05366=1062.623,389.328,386.908,174.818,36.718,156.923
C05367=1062.630,389.575,386.866,174.824,36.725,156.924
C05368=1062.638,389.821,386.826,174.829,36.733,156.926
C05369=1062.646,390.067,386.785,174.835,36.740,156.928
C05370=1062.654,390.314,386.744,174.840,36.747,156.930
C05371=1062.661,390.560,386.703,174.846,36.754,156.931
C05372=1062.668,390.807,386.661,174.851,36.762,156.933
C05373=1062.675,391.054,386.620,174.857,36.769,156.935
C05374=1062.684,391.299,386.579,174.862,36.777,156.937
C05375=1062.691,391.546,386.538,174.868,36.784,156.939
C05376=1062.698,391.792,386.496,174.874,36.792,156.941
C05377=1062.706,392.039,386.456,174.879,36.799,156.942
C05378=1062.714,392.285,386.415,174.885,36.806,156.944
C05379=1062.721,392.531,386.373,174.890,36.814,156.946
C05380=1062.729,392.778,386.331,174.896,36.822,156.948
C05381=1062.737,393.024,386.291,174.902,36.829,156.950
C05382=1062.744,393.270,386.249,174.908,36.837,156.952
C05383=1062.751,393.517,386.208,174.913,36.844,156.953
C05384=1062.759,393.763,386.166,174.919,36.852,156.955
C05385=1062.767,394.010,386.124,174.924,36.860,156.957
C05386=1062.775,394.256,386.082,174.931,36.867,156.959
C05387=1062.782,394.503,386.041,174.936,36.875,156.961
C05388=1062.790,394.748,386.000,174.942,36.882,156.963
C05389=1062.797,394.995,385.958,174.947,36.890,156.965
C05390=1062.805,395.241,385.916,174.954,36.898,156.967
C05391=1062.813,395.487,385.874,174.959,36.906,156.969
C05392=1062.821,395.734,385.833,174.965,36.913,156.970
C05393=1062.828,395.980,385.791,174.970,36.921,156.972
C05394=1062.836,396.226,385.749,174.977,36.929,156.974
C05395=1062.844,396.473,385.707,174.983,36.936,156.976
C05396=1062.851,396.719,385.665,174.988,36.945,156.978
C05397=1062.859,396.965,385.623,174.994,36.952,156.980
C05398=1062.866,397.211,385.581,175.000,36.960,156.982
C05399=1062.875,397.458,385.539,175.006,36.968,156.984
C05400=1062.882,397.704,385.497,175.012,36.976,156.986
C05401=1062.889,397.950,385.456,175.018,36.984,156.988
C05402=1062.898,398.197,385.414,175.024,36.992,156.990
C05403=1062.905,398.443,385.372,175.029,37.000,156.992
C05404=1062.913,398.690,385.329,175.036,37.008,156.994
C05405=1062.921,398.935,385.287,175.042,37.016,156.996
C05406=1062.928,399.181,385.244,175.047,37.024,156.998
C05407=1062.936,399.428,385.202,175.054,37.032,157.000
C05408=1062.944,399.674,385.160,175.060,37.040,157.002
C05409=1062.952,399.921,385.118,175.065,37.048,157.004
C05410=1062.960,400.167,385.076,175.072,37.056,157.006
C05411=1062.968,400.413,385.033,175.078,37.064,157.008
C05412=1062.977,400.717,384.980,175.085,37.074,157.011
C05413=1062.987,401.022,384.928,175.092,37.085,157.013
C05414=1062.997,401.326,384.875,175.100,37.095,157.016
C05415=1063.007,401.631,384.823,175.108,37.105,157.018
C05416=1063.014,401.878,384.780,175.114,37.113,157.020
C05417=1063.022,402.124,384.738,175.121,37.121,157.022
C05418=1063.030,402.370,384.695,175.126,37.130,157.025
C05419=1063.039,402.616,384.652,175.133,37.138,157.027
C05420=1063.046,402.862,384.609,175.139,37.146,157.029
C05421=1063.054,403.109,384.567,175.146,37.155,157.031
C05422=1063.063,403.355,384.524,175.151,37.163,157.033
C05423=1063.069,403.601,384.481,175.157,37.172,157.035
C05424=1063.078,403.847,384.438,175.164,37.180,157.037
C05425=1063.086,404.093,384.395,175.170,37.189,157.039
C05426=1063.093,404.339,384.353,175.177,37.197,157.042
C05427=1063.102,404.585,384.310,175.182,37.205,157.044
C05428=1063.109,404.832,384.266,175.189,37.214,157.046
C05429=1063.118,405.078,384.223,175.195,37.222,157.048
C05430=1063.125,405.324,384.180,175.202,37.231,157.050
C05431=1063.133,405.570,384.137,175.208,37.240,157.053
C05432=1063.141,405.817,384.094,175.215,37.249,157.055
C05433=1063.150,406.063,384.051,175.221,37.257,157.057
C05434=1063.157,406.309,384.007,175.227,37.266,157.059
C05435=1063.165,406.554,383.964,175.234,37.275,157.061
C05436=1063.173,406.801,383.921,175.240,37.283,157.064
C05437=1063.181,407.047,383.877,175.247,37.292,157.066
C05438=1063.190,407.292,383.833,175.253,37.301,157.068
C05439=1063.197,407.539,383.790,175.260,37.309,157.070
C05440=1063.205,407.785,383.746,175.266,37.318,157.073
C05441=1063.214,408.031,383.703,175.273,37.327,157.075
C05442=1063.221,408.277,383.660,175.280,37.336,157.077
C05443=1063.229,408.523,383.616,175.286,37.345,157.079
C05444=1063.237,408.769,383.573,175.293,37.354,157.082
C05445=1063.245,409.015,383.529,175.300,37.363,157.084
C05446=1063.253,409.261,383.485,175.306,37.372,157.086
C05447=1063.262,409.507,383.442,175.313,37.381,157.088
C05448=1063.270,409.753,383.397,175.320,37.390,157.091
C05449=1063.278,409.999,383.354,175.326,37.399,157.093
C05450=1063.285,410.245,383.310,175.333,37.408,157.095
C05451=1063.295,410.492,383.266,175.340,37.417,157.098
C05452=1063.303,410.737,383.222,175.346,37.426,157.100
C05453=1063.311,410.984,383.178,175.353,37.435,157.103
C05454=1063.319,411.229,383.134,175.360,37.444,157.105
C05455=1063.327,411.475,383.091,175.367,37.454,157.107
C05456=1063.335,411.721,383.046,175.374,37.463,157.110
C05457=1063.343,411.967,383.002,175.381,37.472,157.112
